   "Unit1.MotionNodes".PLCToMotion.Parameters.StackMain.StackCalculate.TeachingPos.StartPos.CathodePnPX1 := "Unit1.Em5.Config".cmCathodeMainPnP1AxisX.setPositions[0].position;
   "Unit1.MotionNodes".PLCToMotion.Parameters.StackMain.StackCalculate.TeachingPos.StartPos.CathodePnPX2 := "Unit1.Em5.Config".cmCathodeMainPnP2AxisX.setPositions[0].position;
   "Unit1.MotionNodes".PLCToMotion.Parameters.StackMain.StackCalculate.TeachingPos.StartPos.CathodePnPZ1 := "Unit1.Em5.Config".cmCathodeMainPnP1AxisZ.setPositions[0].position;
   "Unit1.MotionNodes".PLCToMotion.Parameters.StackMain.StackCalculate.TeachingPos.StartPos.CathodePnPZ2 := "Unit1.Em5.Config".cmCathodeMainPnP2AxisZ.setPositions[0].position;

   "Unit1.MotionNodes".PLCToMotion.Parameters.StackMain.StackCalculate.TeachingPos.StartPos.AnodeMandrelYFront := "Unit1.Em6.Config".cmMendrelAnodeFrontAxisY.setPositions[0].position;
   "Unit1.MotionNodes".PLCToMotion.Parameters.StackMain.StackCalculate.TeachingPos.StartPos.AnodeMandrelYRear := "Unit1.Em6.Config".cmMendrelAnodeRearAxisY.setPositions[0].position;
   "Unit1.MotionNodes".PLCToMotion.Parameters.StackMain.StackCalculate.TeachingPos.StartPos.AnodeMandrelZFront := "Unit1.Em6.Config".cmMendrelAnodeFrontAxisZ.setPositions[0].position;
   "Unit1.MotionNodes".PLCToMotion.Parameters.StackMain.StackCalculate.TeachingPos.StartPos.AnodeMandrelZRear := "Unit1.Em6.Config".cmMendrelAnodeRearAxisZ.setPositions[0].position;
   "Unit1.MotionNodes".PLCToMotion.Parameters.StackMain.StackCalculate.TeachingPos.StartPos.CathodeMandrelYFront := "Unit1.Em6.Config".cmMendrelCathodeFrontAxisY.setPositions[0].position;
   "Unit1.MotionNodes".PLCToMotion.Parameters.StackMain.StackCalculate.TeachingPos.StartPos.CathodeMandrelYRear := "Unit1.Em6.Config".cmMendrelCathodeRearAxisY.setPositions[0].position;
   "Unit1.MotionNodes".PLCToMotion.Parameters.StackMain.StackCalculate.TeachingPos.StartPos.CathodeMandrelZFront := "Unit1.Em6.Config".cmMendrelCathodeFrontAxisZ.setPositions[0].position;
   "Unit1.MotionNodes".PLCToMotion.Parameters.StackMain.StackCalculate.TeachingPos.StartPos.CathodeMandrelZRear := "Unit1.Em6.Config".cmMendrelCathodeRearAxisZ.setPositions[0].position;

   ///// End Pos

   "Unit1.MotionNodes".PLCToMotion.Parameters.StackMain.StackCalculate.TeachingPos.EndPos.FinalRoller := "Unit1.Em6.Config".cmFinalRollerFrontAxisX.setPositions[1].position;
   "Unit1.MotionNodes".PLCToMotion.Parameters.StackMain.StackCalculate.TeachingPos.EndPos.AnodePnPX1 := "Unit1.Em4.Config".cmAnodeMainPnP1AxisX.setPositions[1].position;
   "Unit1.MotionNodes".PLCToMotion.Parameters.StackMain.StackCalculate.TeachingPos.EndPos.AnodePnPX2 := "Unit1.Em4.Config".cmAnodeMainPnP2AxisX.setPositions[1].position;

   "Unit1.MotionNodes".PLCToMotion.Parameters.StackMain.StackCalculate.TeachingPos.EndPos.AnodePnPZ1P1 := "Unit1.Em4.Config".cmAnodeMainPnP1AxisZ.setPositions[1].position;
   "Unit1.MotionNodes".PLCToMotion.Parameters.StackMain.StackCalculate.TeachingPos.EndPos.AnodePnPZ1P2 := "Unit1.Em4.Config".cmAnodeMainPnP1AxisZ.setPositions[2].position;
   "Unit1.MotionNodes".PLCToMotion.Parameters.StackMain.StackCalculate.TeachingPos.EndPos.AnodePnPZ2P1 := "Unit1.Em4.Config".cmAnodeMainPnP2AxisZ.setPositions[1].position;
   "Unit1.MotionNodes".PLCToMotion.Parameters.StackMain.StackCalculate.TeachingPos.EndPos.AnodePnPZ2P2 := "Unit1.Em4.Config".cmAnodeMainPnP2AxisZ.setPositions[2].position;

   "Unit1.MotionNodes".PLCToMotion.Parameters.StackMain.StackCalculate.TeachingPos.EndPos.CathodePnPX1 := "Unit1.Em5.Config".cmCathodeMainPnP1AxisX.setPositions[1].position;
   "Unit1.MotionNodes".PLCToMotion.Parameters.StackMain.StackCalculate.TeachingPos.EndPos.CathodePnPX2 := "Unit1.Em5.Config".cmCathodeMainPnP2AxisX.setPositions[1].position;

   "Unit1.MotionNodes".PLCToMotion.Parameters.StackMain.StackCalculate.TeachingPos.EndPos.CathodePnPZ1P1 := "Unit1.Em5.Config".cmCathodeMainPnP1AxisZ.setPositions[1].position;
   "Unit1.MotionNodes".PLCToMotion.Parameters.StackMain.StackCalculate.TeachingPos.EndPos.CathodePnPZ1P2 := "Unit1.Em5.Config".cmCathodeMainPnP1AxisZ.setPositions[2].position;
   "Unit1.MotionNodes".PLCToMotion.Parameters.StackMain.StackCalculate.TeachingPos.EndPos.CathodePnPZ2P1 := "Unit1.Em5.Config".cmCathodeMainPnP2AxisZ.setPositions[1].position;
   "Unit1.MotionNodes".PLCToMotion.Parameters.StackMain.StackCalculate.TeachingPos.EndPos.CathodePnPZ2P2 := "Unit1.Em5.Config".cmCathodeMainPnP2AxisZ.setPositions[2].position;


   "Unit1.MotionNodes".PLCToMotion.Parameters.StackMain.StackCalculate.TeachingPos.EndPos.AnodeMandrelYFront := "Unit1.Em6.Config".cmMendrelAnodeFrontAxisY.setPositions[1].position;
   "Unit1.MotionNodes".PLCToMotion.Parameters.StackMain.StackCalculate.TeachingPos.EndPos.AnodeMandrelYRear := "Unit1.Em6.Config".cmMendrelAnodeRearAxisY.setPositions[1].position;
   "Unit1.MotionNodes".PLCToMotion.Parameters.StackMain.StackCalculate.TeachingPos.EndPos.AnodeMandrelZFront := "Unit1.Em6.Config".cmMendrelAnodeFrontAxisZ.setPositions[1].position;
   "Unit1.MotionNodes".PLCToMotion.Parameters.StackMain.StackCalculate.TeachingPos.EndPos.AnodeMandrelZRear := "Unit1.Em6.Config".cmMendrelAnodeRearAxisZ.setPositions[1].position;
   "Unit1.MotionNodes".PLCToMotion.Parameters.StackMain.StackCalculate.TeachingPos.EndPos.CathodeMandrelYFront := "Unit1.Em6.Config".cmMendrelCathodeFrontAxisY.setPositions[1].position;
   "Unit1.MotionNodes".PLCToMotion.Parameters.StackMain.StackCalculate.TeachingPos.EndPos.CathodeMandrelYRear := "Unit1.Em6.Config".cmMendrelCathodeRearAxisY.setPositions[1].position;
   "Unit1.MotionNodes".PLCToMotion.Parameters.StackMain.StackCalculate.TeachingPos.EndPos.CathodeMandrelZFront := "Unit1.Em6.Config".cmMendrelCathodeFrontAxisZ.setPositions[1].position;
   "Unit1.MotionNodes".PLCToMotion.Parameters.StackMain.StackCalculate.TeachingPos.EndPos.CathodeMandrelZRear := "Unit1.Em6.Config".cmMendrelCathodeRearAxisZ.setPositions[1].position;
END_REGION

REGION Network 8 (SCL): PLC -> HMI Softcam
   "HMI_Interface_Parameter".Softcam[1] := "Unit1.Em0.HmiInterface".cm.softCam.unwinderTopAxisB;
   "HMI_Interface_Parameter".Softcam[2] := "Unit1.Em1.HmiInterface".cm.softCam.unwinderBtmAxisB;
   "HMI_Interface_Parameter".Softcam[3] := "Unit1.Em3.HmiInterface".cm.softCam.compensatorAxisX;
   "HMI_Interface_Parameter".Softcam[4] := "Unit1.Em7.HmiInterface".cm.softCam.jrPusherAxisZ;
   "HMI_Interface_Parameter".Softcam[5] := "Unit1.Em4.HmiInterface".cm.softCam.anodeMainPnP1AxisX;
   "HMI_Interface_Parameter".Softcam[6] := "Unit1.Em4.HmiInterface".cm.softCam.anodeMainPnP2AxisX;
   "HMI_Interface_Parameter".Softcam[7] := "Unit1.Em5.HmiInterface".cm.softCam.cathodeMainPnP1AxisX;
   "HMI_Interface_Parameter".Softcam[8] := "Unit1.Em5.HmiInterface".cm.softCam.cathodeMainPnP2AxisX;
   "HMI_Interface_Parameter".Softcam[9] := "Unit1.Em5.HmiInterface".cm.softCam.cathodeMainPnP1AxisY;
   "HMI_Interface_Parameter".Softcam[10] := "Unit1.Em5.HmiInterface".cm.softCam.cathodeMainPnP1AxisZ;
   "HMI_Interface_Parameter".Softcam[11] := "Unit1.Em4.HmiInterface".cm.softCam.anodeMainPnP1AxisY;
   "HMI_Interface_Parameter".Softcam[12] := "Unit1.Em4.HmiInterface".cm.softCam.anodeMainPnP1AxisZ;
   "HMI_Interface_Parameter".Softcam[13] := "Unit1.Em5.HmiInterface".cm.softCam.cathodeMainPnP2AxisZ;
   "HMI_Interface_Parameter".Softcam[14] := "Unit1.Em4.HmiInterface".cm.softCam.anodeMainPnP2AxisZ;
   "HMI_Interface_Parameter".Softcam[15] := "Unit1.Em4.HmiInterface".cm.softCam.anodeAlignTableAxisX;
   "HMI_Interface_Parameter".Softcam[16] := "Unit1.Em4.HmiInterface".cm.softCam.anodeAlignTableAxisY2;
   "HMI_Interface_Parameter".Softcam[17] := "Unit1.Em4.HmiInterface".cm.softCam.anodeAlignTableAxisY1;
   "HMI_Interface_Parameter".Softcam[18] := "Unit1.Em5.HmiInterface".cm.softCam.cathodeAlignTableAxisX;
   "HMI_Interface_Parameter".Softcam[19] := "Unit1.Em5.HmiInterface".cm.softCam.cathodeAlignTableAxisY2;
   "HMI_Interface_Parameter".Softcam[20] := "Unit1.Em5.HmiInterface".cm.softCam.cathodeAlignTableAxisY1;
   "HMI_Interface_Parameter".Softcam[21] := "Unit1.Em6.HmiInterface".cm.softCam.finalRollerFrontAxisX;
   "HMI_Interface_Parameter".Softcam[22] := "Unit1.Em6.HmiInterface".cm.softCam.finalRollerRearAxisX;
   "HMI_Interface_Parameter".Softcam[23] := "Unit1.Em6.HmiInterface".cm.softCam.mendrelAnodeFrontAxisY;
   "HMI_Interface_Parameter".Softcam[24] := "Unit1.Em6.HmiInterface".cm.softCam.mendrelAnodeFrontAxisZ;
   "HMI_Interface_Parameter".Softcam[25] := "Unit1.Em6.HmiInterface".cm.softCam.mendrelAnodeRearAxisY;
   "HMI_Interface_Parameter".Softcam[26] := "Unit1.Em6.HmiInterface".cm.softCam.mendrelAnodeRearAxisZ;
   "HMI_Interface_Parameter".Softcam[27] := "Unit1.Em6.HmiInterface".cm.softCam.mendrelCathodeFrontAxisY;
   "HMI_Interface_Parameter".Softcam[28] := "Unit1.Em6.HmiInterface".cm.softCam.mendrelCathodeFrontAxisZ;
   "HMI_Interface_Parameter".Softcam[29] := "Unit1.Em6.HmiInterface".cm.softCam.mendrelCathodeRearAxisY;
   "HMI_Interface_Parameter".Softcam[30] := "Unit1.Em6.HmiInterface".cm.softCam.mendrelCathodeRearAxisZ;
   "HMI_Interface_Parameter".Softcam[31] := "Unit1.Em6.HmiInterface".cm.softCam.stackTableAxisZ;
   "HMI_Interface_Parameter".Softcam[32] := "Unit1.Em6.HmiInterface".cm.softCam.stackTableOutFrontAxisZ;
   "HMI_Interface_Parameter".Softcam[33] := "Unit1.Em6.HmiInterface".cm.softCam.stackTableOutRearAxisZ;
   "HMI_Interface_Parameter".Softcam[34] := "Unit1.Em7.HmiInterface".cm.softCam.sepaClampnCutterAxisX;
   "HMI_Interface_Parameter".Softcam[35] := "Unit1.Em7.HmiInterface".cm.softCam.sepaClampnCutterAxisZ;
   "HMI_Interface_Parameter".Softcam[36] := "Unit1.Em7.HmiInterface".cm.softCam.sepaGripperAxisX;
   "HMI_Interface_Parameter".Softcam[37] := "Unit1.Em7.HmiInterface".cm.softCam.sepaGripperAxisZ;
   "HMI_Interface_Parameter".Softcam[38] := "Unit1.Em7.HmiInterface".cm.softCam.sepaGripperAxisC;
   "HMI_Interface_Parameter".Softcam[39] := "Unit1.Em7.HmiInterface".cm.softCam.jrWinderRearAxisY;
   "HMI_Interface_Parameter".Softcam[40] := "Unit1.Em7.HmiInterface".cm.softCam.jrWinderFrontAxisY;
   "HMI_Interface_Parameter".Softcam[41] := "Unit1.Em7.HmiInterface".cm.softCam.jrWinderAxisB;
END_REGION

REGION Network 9 (SCL): SamplingMode Complete end
   IF "Unit1.EmNodes".SamplingModeComplete THEN
       "HMI_Interface_Parameter".FATModeInterface.ModeSelect.SamplingMode := FALSE;
       ;
   END_IF;
END_REGION

REGION Network 10: SamplingMode Btn on count reset trigger // cell current count
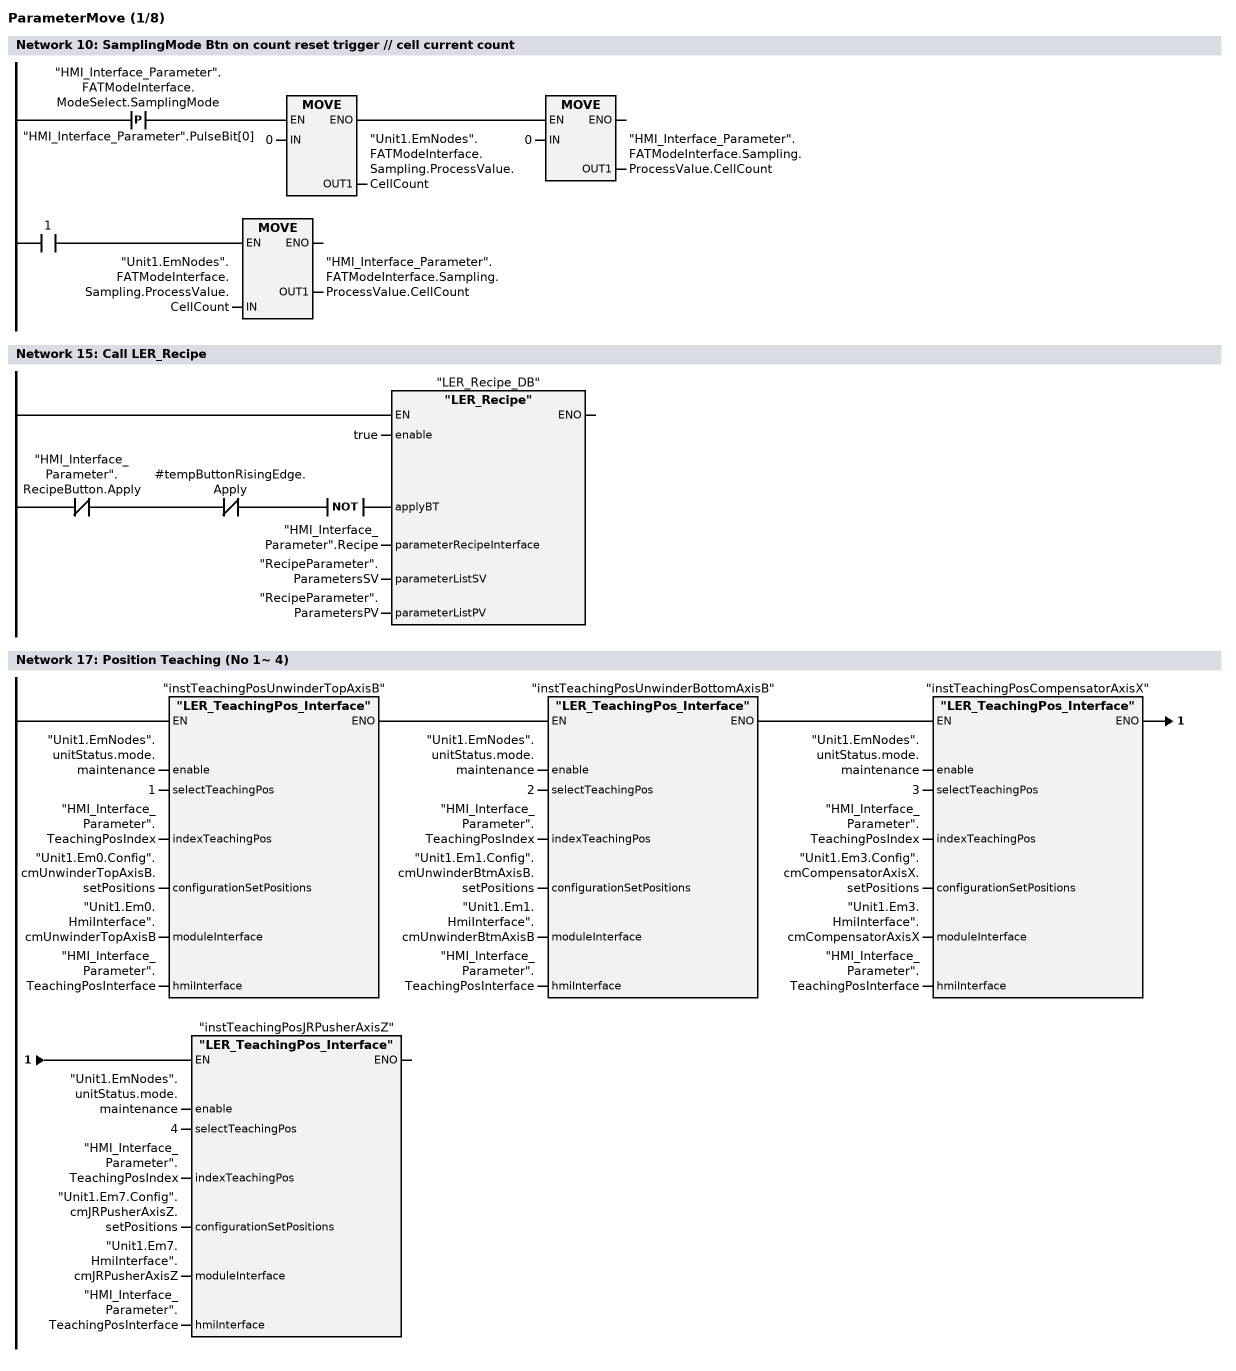
   RUNG wire#powerrail
      P_Contact(operand := "HMI_Interface_Parameter".FATModeInterface.ModeSelect.SamplingMode, bit := "HMI_Interface_Parameter".PulseBit[0])
      Move(in := 0, out1 => "Unit1.EmNodes".FATModeInterface.Sampling.ProcessValue.CellCount)
      Move(in := 0, out1 => "HMI_Interface_Parameter".FATModeInterface.Sampling.ProcessValue.CellCount)
   END_RUNG
   RUNG wire#powerrail
      Contact( 1 )
      Move(in := "Unit1.EmNodes".FATModeInterface.Sampling.ProcessValue.CellCount, out1 => "HMI_Interface_Parameter".FATModeInterface.Sampling.ProcessValue.CellCount)
   END_RUNG
   // the same network as SCL:
   #_w1 := "HMI_Interface_Parameter".FATModeInterface.ModeSelect.SamplingMode AND NOT "HMI_Interface_Parameter".PulseBit[0];   // rising edge of "HMI_Interface_Parameter".FATModeInterface.ModeSelect.SamplingMode
   "HMI_Interface_Parameter".PulseBit[0] := "HMI_Interface_Parameter".FATModeInterface.ModeSelect.SamplingMode;
   IF #_w1 THEN
       "Unit1.EmNodes".FATModeInterface.Sampling.ProcessValue.CellCount := 0;
       "HMI_Interface_Parameter".FATModeInterface.Sampling.ProcessValue.CellCount := 0;
   END_IF;
   IF 1 THEN
       "HMI_Interface_Parameter".FATModeInterface.Sampling.ProcessValue.CellCount := "Unit1.EmNodes".FATModeInterface.Sampling.ProcessValue.CellCount;
   END_IF;
END_REGION

REGION Network 12 (SCL): HMI Interface Parameter To Recipe Pareameter SV
   // IF #tempButtonRisingEdge.Apply THEN
   //     "RecipeParameter".ParametersSV.Recipe1 := "HMI_Interface_Parameter"."Default Recipe".SetValue."Electrode Width".Anode;
   //     "RecipeParameter".ParametersSV.Recipe2 := "HMI_Interface_Parameter"."Default Recipe".SetValue."Electrode Width".Cathode;
   //     "RecipeParameter".ParametersSV.Recipe3 := "HMI_Interface_Parameter"."Default Recipe".SetValue."Anode Thinkness";
   //     "RecipeParameter".ParametersSV.Recipe4 := "HMI_Interface_Parameter"."Default Recipe".SetValue."Cathode Thinkness";
   //     "RecipeParameter".ParametersSV.Recipe5 := "HMI_Interface_Parameter"."Default Recipe".SetValue."Sperator Thinkness";
   //     "RecipeParameter".ParametersSV.Recipe6 := "HMI_Interface_Parameter"."Default Recipe".SetValue."Jelly Roll Width";
   //     "RecipeParameter".ParametersSV.Recipe7 := "HMI_Interface_Parameter"."Default Recipe".SetValue."Cell Stack Count";
   //     "RecipeParameter".ParametersSV.Recipe8 := "HMI_Interface_Parameter".Parameter_Image[0]."Set Value";
   //     "RecipeParameter".ParametersSV.Recipe9 := "HMI_Interface_Parameter".Parameter_Image[1]."Set Value";
   //     //
   //     //"RecipeParameter".ParametersSV.Recipe10 := ;
   //     //"RecipeParameter".ParametersSV.Recipe11 := ;
   //     //"RecipeParameter".ParametersSV.Recipe12 := ;
   //     //"RecipeParameter".ParametersSV.Recipe13 := ;
   //     //"RecipeParameter".ParametersSV.Recipe14 := ;
   //     //"RecipeParameter".ParametersSV.Recipe15 := ;
   //     //"RecipeParameter".ParametersSV.Recipe16 := ;
   //     //"RecipeParameter".ParametersSV.Recipe17 := ;
   //     //"RecipeParameter".ParametersSV.Recipe18 := ;
   //     //"RecipeParameter".ParametersSV.Recipe19 := ;
   //     //"RecipeParameter".ParametersSV.Recipe20 := ;
   //     //"RecipeParameter".ParametersSV.Recipe21 := ;
   //     //"RecipeParameter".ParametersSV.Recipe22 := ;
   //     //"RecipeParameter".ParametersSV.Recipe23 := ;
   //     //"RecipeParameter".ParametersSV.Recipe24 := ;
   //     //"RecipeParameter".ParametersSV.Recipe25 := ;
   // END_IF;
END_REGION

REGION Network 13 (SCL): HMI Interface Pareameter Recipe Data To HMI Interface Parameter Process Value
   // IF "HMI_Interface_Parameter".Recipe.RecipeChangeBT OR "HMI_Interface_Parameter".RecipeButton.Apply OR #tempButtonRisingEdge.Apply THEN

   //     "HMI_Interface_Parameter"."Default Recipe".ProcessValue."Electrode Width".Anode := "HMI_Interface_Parameter".Recipe.Recipe_Data["HMI_Interface_Parameter".Recipe.CurrentRecipeNum].Recipe1;
   //     "HMI_Interface_Parameter"."Default Recipe".ProcessValue."Electrode Width".Cathode := "HMI_Interface_Parameter".Recipe.Recipe_Data["HMI_Interface_Parameter".Recipe.CurrentRecipeNum].Recipe2;
   //     "HMI_Interface_Parameter"."Default Recipe".ProcessValue."Anode Thinkness" := "HMI_Interface_Parameter".Recipe.Recipe_Data["HMI_Interface_Parameter".Recipe.CurrentRecipeNum].Recipe3;
   //     "HMI_Interface_Parameter"."Default Recipe".ProcessValue."Cathode Thinkness" := "HMI_Interface_Parameter".Recipe.Recipe_Data["HMI_Interface_Parameter".Recipe.CurrentRecipeNum].Recipe4;
   //     "HMI_Interface_Parameter"."Default Recipe".ProcessValue."Sperator Thinkness" := "HMI_Interface_Parameter".Recipe.Recipe_Data["HMI_Interface_Parameter".Recipe.CurrentRecipeNum].Recipe5;
   //     "HMI_Interface_Parameter"."Default Recipe".ProcessValue."Jelly Roll Width" := "HMI_Interface_Parameter".Recipe.Recipe_Data["HMI_Interface_Parameter".Recipe.CurrentRecipeNum].Recipe6;
   //     "HMI_Interface_Parameter"."Default Recipe".ProcessValue."Cell Stack Count" := LREAL_TO_SINT("HMI_Interface_Parameter".Recipe.Recipe_Data["HMI_Interface_Parameter".Recipe.CurrentRecipeNum].Recipe7);
   //     "HMI_Interface_Parameter".Parameter_Image[0]."Process Value" := "HMI_Interface_Parameter".Recipe.Recipe_Data["HMI_Interface_Parameter".Recipe.CurrentRecipeNum].Recipe8;
   //     "HMI_Interface_Parameter".Parameter_Image[1]."Process Value" := "HMI_Interface_Parameter".Recipe.Recipe_Data["HMI_Interface_Parameter".Recipe.CurrentRecipeNum].Recipe9;
   //     // := "HMI_Interface_Parameter".Recipe.Recipe_Data["HMI_Interface_Parameter".Recipe.CurrentRecipeNum].Recipe10;
   //     // := "HMI_Interface_Parameter".Recipe.Recipe_Data["HMI_Interface_Parameter".Recipe.CurrentRecipeNum].Recipe11;
   //     // := "HMI_Interface_Parameter".Recipe.Recipe_Data["HMI_Interface_Parameter".Recipe.CurrentRecipeNum].Recipe12;
   //     // := "HMI_Interface_Parameter".Recipe.Recipe_Data["HMI_Interface_Parameter".Recipe.CurrentRecipeNum].Recipe13;
   //     // := "HMI_Interface_Parameter".Recipe.Recipe_Data["HMI_Interface_Parameter".Recipe.CurrentRecipeNum].Recipe14;
   //     // := "HMI_Interface_Parameter".Recipe.Recipe_Data["HMI_Interface_Parameter".Recipe.CurrentRecipeNum].Recipe15;
   // END_IF;
END_REGION

REGION Network 14 (SCL): Recipe Parameter PV To Unit EmData Recipe
   "Unit1.EmData".UnitRecipe.size.Anode.length := "RecipeParameter".ParametersPV.Recipe1;
   "Unit1.EmData".UnitRecipe.size.Cathode.length := "RecipeParameter".ParametersPV.Recipe2;
   "Unit1.EmData".UnitRecipe.size.Anode.thickness := "RecipeParameter".ParametersPV.Recipe3;
   "Unit1.EmData".UnitRecipe.size.Cathode.thickness := "RecipeParameter".ParametersPV.Recipe4;
   "Unit1.EmData".UnitRecipe.SepaThickness := "RecipeParameter".ParametersPV.Recipe5;
   "Unit1.EmData".UnitRecipe.JellyRollWidth := "RecipeParameter".ParametersPV.Recipe6;
   "Unit1.EmData".UnitRecipe.StackCount := "RecipeParameter".ParametersPV.Recipe7;
   "Unit1.EmData".UnitRecipe.DancerRegulator := "RecipeParameter".ParametersPV.Recipe8;
   "Unit1.EmData".UnitRecipe.AutoSpliceRemainingLength := "RecipeParameter".ParametersPV.Recipe9;
   //
   // := "RecipeParameter".ParametersPV.Recipe10;
   // := "RecipeParameter".ParametersPV.Recipe11;
   // := "RecipeParameter".ParametersPV.Recipe12;
   // := "RecipeParameter".ParametersPV.Recipe13;
   // := "RecipeParameter".ParametersPV.Recipe14;
   // := "RecipeParameter".ParametersPV.Recipe15;
END_REGION

REGION Network 15: Call LER_Recipe
   RUNG wire#powerrail
      "LER_Recipe_DB"(applyBT := wire#w1, enable := true, parameterRecipeInterface := "HMI_Interface_Parameter".Recipe, parameterListSV := "RecipeParameter".ParametersSV, parameterListPV := "RecipeParameter".ParametersPV)
   END_RUNG
   RUNG wire#powerrail
      I_Contact( "HMI_Interface_Parameter".RecipeButton.Apply )
      I_Contact( #tempButtonRisingEdge.Apply )
      Not()
   END_RUNG wire#w1
   // the same network as SCL:
   "LER_Recipe_DB"(enable := true,   // "LER_Recipe"
                   applyBT := NOT (NOT "HMI_Interface_Parameter".RecipeButton.Apply AND NOT #tempButtonRisingEdge.Apply),
                   parameterRecipeInterface := "HMI_Interface_Parameter".Recipe,
                   parameterListSV := "RecipeParameter".ParametersSV,
                   parameterListPV := "RecipeParameter".ParametersPV);
END_REGION

REGION Network 17: Position Teaching (No 1~ 4)
   RUNG wire#powerrail
      "instTeachingPosUnwinderTopAxisB"(enable := "Unit1.EmNodes".unitStatus.mode.maintenance, selectTeachingPos := 1, indexTeachingPos := "HMI_Interface_Parameter".TeachingPosIndex, configurationSetPositions := "Unit1.Em0.Config".cmUnwinderTopAxisB.setPositions, moduleInterface := "Unit1.Em0.HmiInterface".cmUnwinderTopAxisB, hmiInterface := "HMI_Interface_Parameter".TeachingPosInterface)
      "instTeachingPosUnwinderBottomAxisB"(enable := "Unit1.EmNodes".unitStatus.mode.maintenance, selectTeachingPos := 2, indexTeachingPos := "HMI_Interface_Parameter".TeachingPosIndex, configurationSetPositions := "Unit1.Em1.Config".cmUnwinderBtmAxisB.setPositions, moduleInterface := "Unit1.Em1.HmiInterface".cmUnwinderBtmAxisB, hmiInterface := "HMI_Interface_Parameter".TeachingPosInterface)
      "instTeachingPosCompensatorAxisX"(enable := "Unit1.EmNodes".unitStatus.mode.maintenance, selectTeachingPos := 3, indexTeachingPos := "HMI_Interface_Parameter".TeachingPosIndex, configurationSetPositions := "Unit1.Em3.Config".cmCompensatorAxisX.setPositions, moduleInterface := "Unit1.Em3.HmiInterface".cmCompensatorAxisX, hmiInterface := "HMI_Interface_Parameter".TeachingPosInterface)
      "instTeachingPosJRPusherAxisZ"(enable := "Unit1.EmNodes".unitStatus.mode.maintenance, selectTeachingPos := 4, indexTeachingPos := "HMI_Interface_Parameter".TeachingPosIndex, configurationSetPositions := "Unit1.Em7.Config".cmJRPusherAxisZ.setPositions, moduleInterface := "Unit1.Em7.HmiInterface".cmJRPusherAxisZ, hmiInterface := "HMI_Interface_Parameter".TeachingPosInterface)
   END_RUNG
   // the same network as SCL:
   "instTeachingPosUnwinderTopAxisB"(enable := "Unit1.EmNodes".unitStatus.mode.maintenance,   // "LER_TeachingPos_Interface"
                           selectTeachingPos := 1,
                           indexTeachingPos := "HMI_Interface_Parameter".TeachingPosIndex,
                           configurationSetPositions := "Unit1.Em0.Config".cmUnwinderTopAxisB.setPositions,
                           moduleInterface := "Unit1.Em0.HmiInterface".cmUnwinderTopAxisB,
                           hmiInterface := "HMI_Interface_Parameter".TeachingPosInterface,
                           ENO => #_w1);
   "instTeachingPosUnwinderBottomAxisB"(EN := #_w1,   // "LER_TeachingPos_Interface"
                           enable := "Unit1.EmNodes".unitStatus.mode.maintenance,
                           selectTeachingPos := 2,
                           indexTeachingPos := "HMI_Interface_Parameter".TeachingPosIndex,
                           configurationSetPositions := "Unit1.Em1.Config".cmUnwinderBtmAxisB.setPositions,
                           moduleInterface := "Unit1.Em1.HmiInterface".cmUnwinderBtmAxisB,
                           hmiInterface := "HMI_Interface_Parameter".TeachingPosInterface,
                           ENO => #_w2);
   "instTeachingPosCompensatorAxisX"(EN := #_w2,   // "LER_TeachingPos_Interface"
                           enable := "Unit1.EmNodes".unitStatus.mode.maintenance,
                           selectTeachingPos := 3,
                           indexTeachingPos := "HMI_Interface_Parameter".TeachingPosIndex,
                           configurationSetPositions := "Unit1.Em3.Config".cmCompensatorAxisX.setPositions,
                           moduleInterface := "Unit1.Em3.HmiInterface".cmCompensatorAxisX,
                           hmiInterface := "HMI_Interface_Parameter".TeachingPosInterface,
                           ENO => #_w3);
   IF #_w3 THEN
       "instTeachingPosJRPusherAxisZ"(enable := "Unit1.EmNodes".unitStatus.mode.maintenance,   // "LER_TeachingPos_Interface"
                               selectTeachingPos := 4,
                               indexTeachingPos := "HMI_Interface_Parameter".TeachingPosIndex,
                               configurationSetPositions := "Unit1.Em7.Config".cmJRPusherAxisZ.setPositions,
                               moduleInterface := "Unit1.Em7.HmiInterface".cmJRPusherAxisZ,
                               hmiInterface := "HMI_Interface_Parameter".TeachingPosInterface);
   END_IF;
END_REGION

REGION Network 18: Position Teaching (No 5~8)
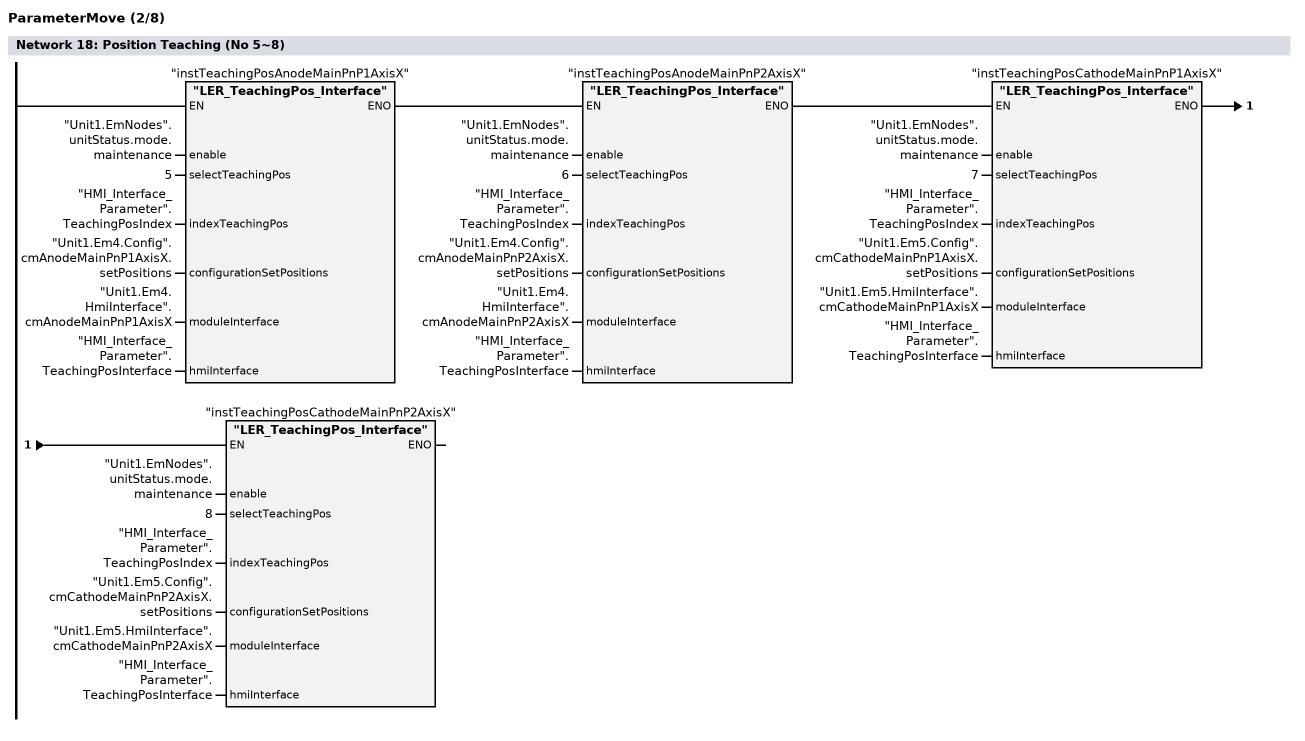
   RUNG wire#powerrail
      "instTeachingPosAnodeMainPnP1AxisX"(enable := "Unit1.EmNodes".unitStatus.mode.maintenance, selectTeachingPos := 5, indexTeachingPos := "HMI_Interface_Parameter".TeachingPosIndex, configurationSetPositions := "Unit1.Em4.Config".cmAnodeMainPnP1AxisX.setPositions, moduleInterface := "Unit1.Em4.HmiInterface".cmAnodeMainPnP1AxisX, hmiInterface := "HMI_Interface_Parameter".TeachingPosInterface)
      "instTeachingPosAnodeMainPnP2AxisX"(enable := "Unit1.EmNodes".unitStatus.mode.maintenance, selectTeachingPos := 6, indexTeachingPos := "HMI_Interface_Parameter".TeachingPosIndex, configurationSetPositions := "Unit1.Em4.Config".cmAnodeMainPnP2AxisX.setPositions, moduleInterface := "Unit1.Em4.HmiInterface".cmAnodeMainPnP2AxisX, hmiInterface := "HMI_Interface_Parameter".TeachingPosInterface)
      "instTeachingPosCathodeMainPnP1AxisX"(enable := "Unit1.EmNodes".unitStatus.mode.maintenance, selectTeachingPos := 7, indexTeachingPos := "HMI_Interface_Parameter".TeachingPosIndex, configurationSetPositions := "Unit1.Em5.Config".cmCathodeMainPnP1AxisX.setPositions, moduleInterface := "Unit1.Em5.HmiInterface".cmCathodeMainPnP1AxisX, hmiInterface := "HMI_Interface_Parameter".TeachingPosInterface)
      "instTeachingPosCathodeMainPnP2AxisX"(enable := "Unit1.EmNodes".unitStatus.mode.maintenance, selectTeachingPos := 8, indexTeachingPos := "HMI_Interface_Parameter".TeachingPosIndex, configurationSetPositions := "Unit1.Em5.Config".cmCathodeMainPnP2AxisX.setPositions, moduleInterface := "Unit1.Em5.HmiInterface".cmCathodeMainPnP2AxisX, hmiInterface := "HMI_Interface_Parameter".TeachingPosInterface)
   END_RUNG
   // the same network as SCL:
   "instTeachingPosAnodeMainPnP1AxisX"(enable := "Unit1.EmNodes".unitStatus.mode.maintenance,   // "LER_TeachingPos_Interface"
                           selectTeachingPos := 5,
                           indexTeachingPos := "HMI_Interface_Parameter".TeachingPosIndex,
                           configurationSetPositions := "Unit1.Em4.Config".cmAnodeMainPnP1AxisX.setPositions,
                           moduleInterface := "Unit1.Em4.HmiInterface".cmAnodeMainPnP1AxisX,
                           hmiInterface := "HMI_Interface_Parameter".TeachingPosInterface,
                           ENO => #_w1);
   "instTeachingPosAnodeMainPnP2AxisX"(EN := #_w1,   // "LER_TeachingPos_Interface"
                           enable := "Unit1.EmNodes".unitStatus.mode.maintenance,
                           selectTeachingPos := 6,
                           indexTeachingPos := "HMI_Interface_Parameter".TeachingPosIndex,
                           configurationSetPositions := "Unit1.Em4.Config".cmAnodeMainPnP2AxisX.setPositions,
                           moduleInterface := "Unit1.Em4.HmiInterface".cmAnodeMainPnP2AxisX,
                           hmiInterface := "HMI_Interface_Parameter".TeachingPosInterface,
                           ENO => #_w2);
   "instTeachingPosCathodeMainPnP1AxisX"(EN := #_w2,   // "LER_TeachingPos_Interface"
                           enable := "Unit1.EmNodes".unitStatus.mode.maintenance,
                           selectTeachingPos := 7,
                           indexTeachingPos := "HMI_Interface_Parameter".TeachingPosIndex,
                           configurationSetPositions := "Unit1.Em5.Config".cmCathodeMainPnP1AxisX.setPositions,
                           moduleInterface := "Unit1.Em5.HmiInterface".cmCathodeMainPnP1AxisX,
                           hmiInterface := "HMI_Interface_Parameter".TeachingPosInterface,
                           ENO => #_w3);
   IF #_w3 THEN
       "instTeachingPosCathodeMainPnP2AxisX"(enable := "Unit1.EmNodes".unitStatus.mode.maintenance,   // "LER_TeachingPos_Interface"
                               selectTeachingPos := 8,
                               indexTeachingPos := "HMI_Interface_Parameter".TeachingPosIndex,
                               configurationSetPositions := "Unit1.Em5.Config".cmCathodeMainPnP2AxisX.setPositions,
                               moduleInterface := "Unit1.Em5.HmiInterface".cmCathodeMainPnP2AxisX,
                               hmiInterface := "HMI_Interface_Parameter".TeachingPosInterface);
   END_IF;
END_REGION

REGION Network 19: Position Teaching (No 9~12)
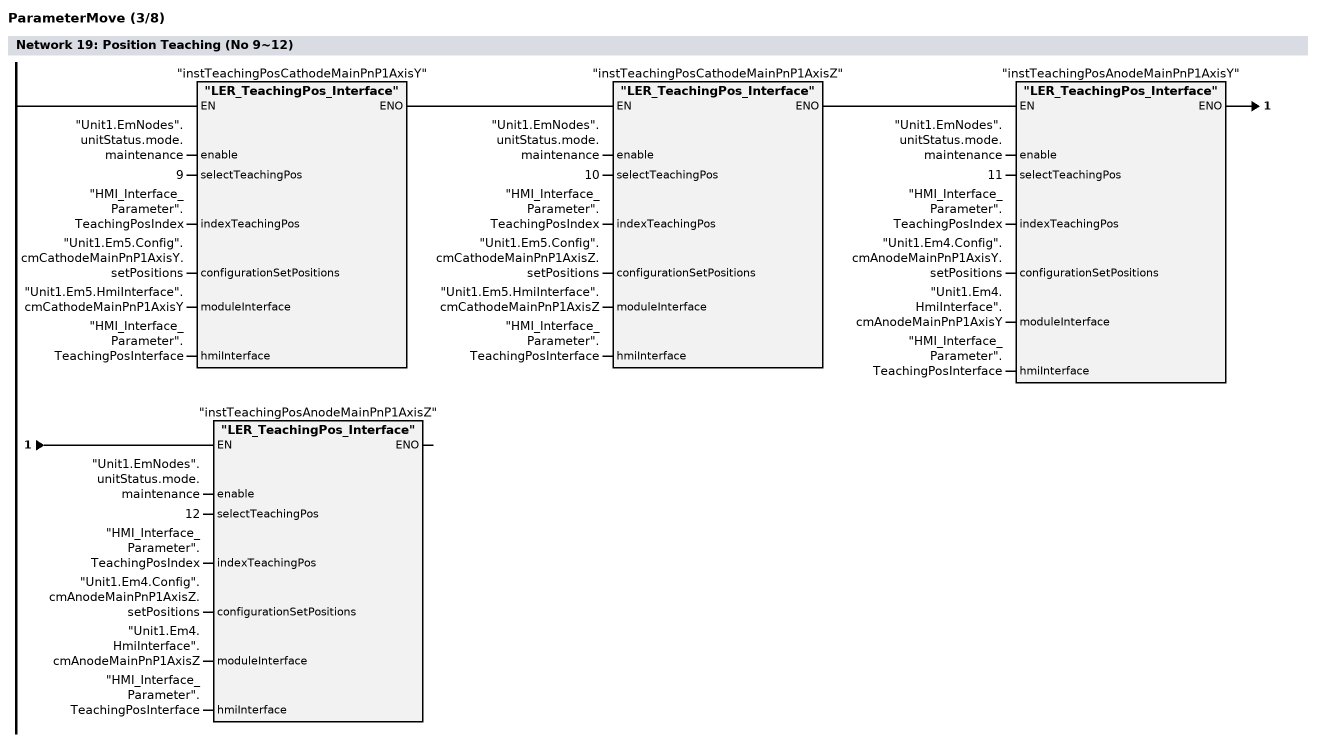
   RUNG wire#powerrail
      "instTeachingPosCathodeMainPnP1AxisY"(enable := "Unit1.EmNodes".unitStatus.mode.maintenance, selectTeachingPos := 9, indexTeachingPos := "HMI_Interface_Parameter".TeachingPosIndex, configurationSetPositions := "Unit1.Em5.Config".cmCathodeMainPnP1AxisY.setPositions, moduleInterface := "Unit1.Em5.HmiInterface".cmCathodeMainPnP1AxisY, hmiInterface := "HMI_Interface_Parameter".TeachingPosInterface)
      "instTeachingPosCathodeMainPnP1AxisZ"(enable := "Unit1.EmNodes".unitStatus.mode.maintenance, selectTeachingPos := 10, indexTeachingPos := "HMI_Interface_Parameter".TeachingPosIndex, configurationSetPositions := "Unit1.Em5.Config".cmCathodeMainPnP1AxisZ.setPositions, moduleInterface := "Unit1.Em5.HmiInterface".cmCathodeMainPnP1AxisZ, hmiInterface := "HMI_Interface_Parameter".TeachingPosInterface)
      "instTeachingPosAnodeMainPnP1AxisY"(enable := "Unit1.EmNodes".unitStatus.mode.maintenance, selectTeachingPos := 11, indexTeachingPos := "HMI_Interface_Parameter".TeachingPosIndex, configurationSetPositions := "Unit1.Em4.Config".cmAnodeMainPnP1AxisY.setPositions, moduleInterface := "Unit1.Em4.HmiInterface".cmAnodeMainPnP1AxisY, hmiInterface := "HMI_Interface_Parameter".TeachingPosInterface)
      "instTeachingPosAnodeMainPnP1AxisZ"(enable := "Unit1.EmNodes".unitStatus.mode.maintenance, selectTeachingPos := 12, indexTeachingPos := "HMI_Interface_Parameter".TeachingPosIndex, configurationSetPositions := "Unit1.Em4.Config".cmAnodeMainPnP1AxisZ.setPositions, moduleInterface := "Unit1.Em4.HmiInterface".cmAnodeMainPnP1AxisZ, hmiInterface := "HMI_Interface_Parameter".TeachingPosInterface)
   END_RUNG
   // the same network as SCL:
   "instTeachingPosCathodeMainPnP1AxisY"(enable := "Unit1.EmNodes".unitStatus.mode.maintenance,   // "LER_TeachingPos_Interface"
                           selectTeachingPos := 9,
                           indexTeachingPos := "HMI_Interface_Parameter".TeachingPosIndex,
                           configurationSetPositions := "Unit1.Em5.Config".cmCathodeMainPnP1AxisY.setPositions,
                           moduleInterface := "Unit1.Em5.HmiInterface".cmCathodeMainPnP1AxisY,
                           hmiInterface := "HMI_Interface_Parameter".TeachingPosInterface,
                           ENO => #_w1);
   "instTeachingPosCathodeMainPnP1AxisZ"(EN := #_w1,   // "LER_TeachingPos_Interface"
                           enable := "Unit1.EmNodes".unitStatus.mode.maintenance,
                           selectTeachingPos := 10,
                           indexTeachingPos := "HMI_Interface_Parameter".TeachingPosIndex,
                           configurationSetPositions := "Unit1.Em5.Config".cmCathodeMainPnP1AxisZ.setPositions,
                           moduleInterface := "Unit1.Em5.HmiInterface".cmCathodeMainPnP1AxisZ,
                           hmiInterface := "HMI_Interface_Parameter".TeachingPosInterface,
                           ENO => #_w2);
   "instTeachingPosAnodeMainPnP1AxisY"(EN := #_w2,   // "LER_TeachingPos_Interface"
                           enable := "Unit1.EmNodes".unitStatus.mode.maintenance,
                           selectTeachingPos := 11,
                           indexTeachingPos := "HMI_Interface_Parameter".TeachingPosIndex,
                           configurationSetPositions := "Unit1.Em4.Config".cmAnodeMainPnP1AxisY.setPositions,
                           moduleInterface := "Unit1.Em4.HmiInterface".cmAnodeMainPnP1AxisY,
                           hmiInterface := "HMI_Interface_Parameter".TeachingPosInterface,
                           ENO => #_w3);
   IF #_w3 THEN
       "instTeachingPosAnodeMainPnP1AxisZ"(enable := "Unit1.EmNodes".unitStatus.mode.maintenance,   // "LER_TeachingPos_Interface"
                               selectTeachingPos := 12,
                               indexTeachingPos := "HMI_Interface_Parameter".TeachingPosIndex,
                               configurationSetPositions := "Unit1.Em4.Config".cmAnodeMainPnP1AxisZ.setPositions,
                               moduleInterface := "Unit1.Em4.HmiInterface".cmAnodeMainPnP1AxisZ,
                               hmiInterface := "HMI_Interface_Parameter".TeachingPosInterface);
   END_IF;
END_REGION

REGION Network 20: Position Teaching (No 13~16)
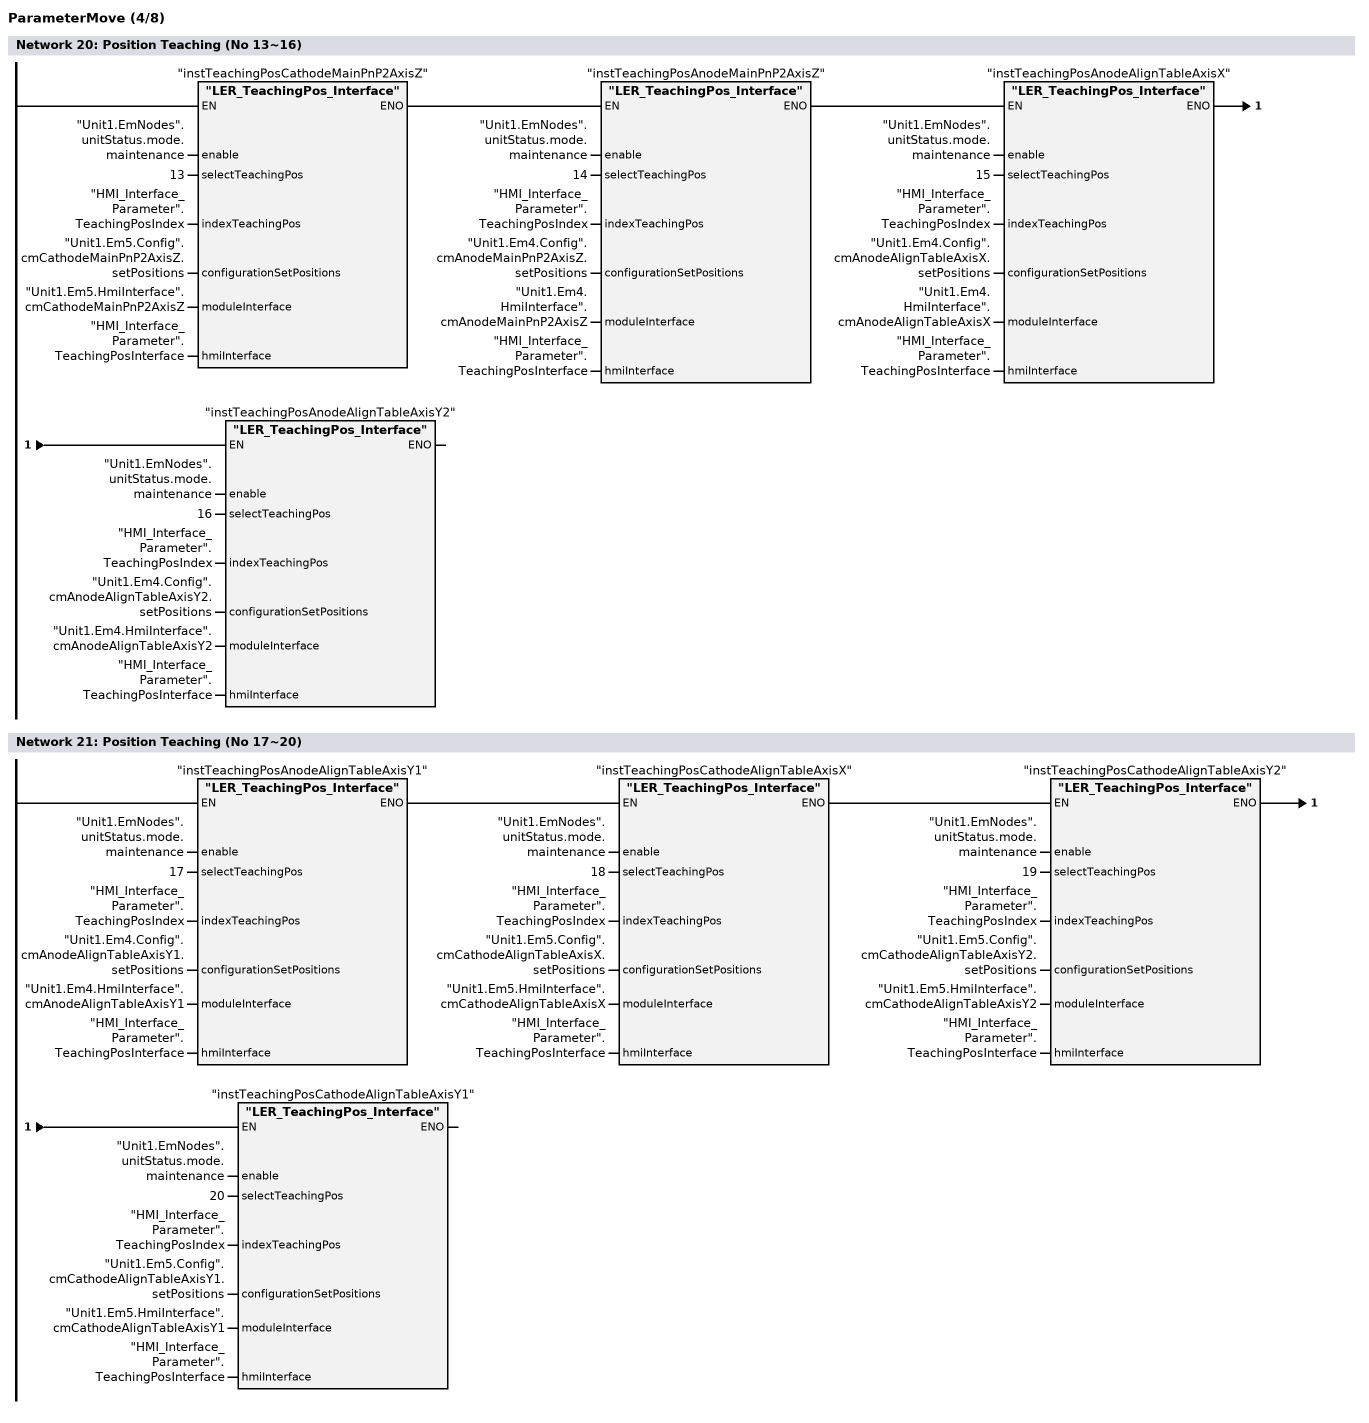
   RUNG wire#powerrail
      "instTeachingPosCathodeMainPnP2AxisZ"(enable := "Unit1.EmNodes".unitStatus.mode.maintenance, selectTeachingPos := 13, indexTeachingPos := "HMI_Interface_Parameter".TeachingPosIndex, configurationSetPositions := "Unit1.Em5.Config".cmCathodeMainPnP2AxisZ.setPositions, moduleInterface := "Unit1.Em5.HmiInterface".cmCathodeMainPnP2AxisZ, hmiInterface := "HMI_Interface_Parameter".TeachingPosInterface)
      "instTeachingPosAnodeMainPnP2AxisZ"(enable := "Unit1.EmNodes".unitStatus.mode.maintenance, selectTeachingPos := 14, indexTeachingPos := "HMI_Interface_Parameter".TeachingPosIndex, configurationSetPositions := "Unit1.Em4.Config".cmAnodeMainPnP2AxisZ.setPositions, moduleInterface := "Unit1.Em4.HmiInterface".cmAnodeMainPnP2AxisZ, hmiInterface := "HMI_Interface_Parameter".TeachingPosInterface)
      "instTeachingPosAnodeAlignTableAxisX"(enable := "Unit1.EmNodes".unitStatus.mode.maintenance, selectTeachingPos := 15, indexTeachingPos := "HMI_Interface_Parameter".TeachingPosIndex, configurationSetPositions := "Unit1.Em4.Config".cmAnodeAlignTableAxisX.setPositions, moduleInterface := "Unit1.Em4.HmiInterface".cmAnodeAlignTableAxisX, hmiInterface := "HMI_Interface_Parameter".TeachingPosInterface)
      "instTeachingPosAnodeAlignTableAxisY2"(enable := "Unit1.EmNodes".unitStatus.mode.maintenance, selectTeachingPos := 16, indexTeachingPos := "HMI_Interface_Parameter".TeachingPosIndex, configurationSetPositions := "Unit1.Em4.Config".cmAnodeAlignTableAxisY2.setPositions, moduleInterface := "Unit1.Em4.HmiInterface".cmAnodeAlignTableAxisY2, hmiInterface := "HMI_Interface_Parameter".TeachingPosInterface)
   END_RUNG
   // the same network as SCL:
   "instTeachingPosCathodeMainPnP2AxisZ"(enable := "Unit1.EmNodes".unitStatus.mode.maintenance,   // "LER_TeachingPos_Interface"
                           selectTeachingPos := 13,
                           indexTeachingPos := "HMI_Interface_Parameter".TeachingPosIndex,
                           configurationSetPositions := "Unit1.Em5.Config".cmCathodeMainPnP2AxisZ.setPositions,
                           moduleInterface := "Unit1.Em5.HmiInterface".cmCathodeMainPnP2AxisZ,
                           hmiInterface := "HMI_Interface_Parameter".TeachingPosInterface,
                           ENO => #_w1);
   "instTeachingPosAnodeMainPnP2AxisZ"(EN := #_w1,   // "LER_TeachingPos_Interface"
                           enable := "Unit1.EmNodes".unitStatus.mode.maintenance,
                           selectTeachingPos := 14,
                           indexTeachingPos := "HMI_Interface_Parameter".TeachingPosIndex,
                           configurationSetPositions := "Unit1.Em4.Config".cmAnodeMainPnP2AxisZ.setPositions,
                           moduleInterface := "Unit1.Em4.HmiInterface".cmAnodeMainPnP2AxisZ,
                           hmiInterface := "HMI_Interface_Parameter".TeachingPosInterface,
                           ENO => #_w2);
   "instTeachingPosAnodeAlignTableAxisX"(EN := #_w2,   // "LER_TeachingPos_Interface"
                           enable := "Unit1.EmNodes".unitStatus.mode.maintenance,
                           selectTeachingPos := 15,
                           indexTeachingPos := "HMI_Interface_Parameter".TeachingPosIndex,
                           configurationSetPositions := "Unit1.Em4.Config".cmAnodeAlignTableAxisX.setPositions,
                           moduleInterface := "Unit1.Em4.HmiInterface".cmAnodeAlignTableAxisX,
                           hmiInterface := "HMI_Interface_Parameter".TeachingPosInterface,
                           ENO => #_w3);
   IF #_w3 THEN
       "instTeachingPosAnodeAlignTableAxisY2"(enable := "Unit1.EmNodes".unitStatus.mode.maintenance,   // "LER_TeachingPos_Interface"
                               selectTeachingPos := 16,
                               indexTeachingPos := "HMI_Interface_Parameter".TeachingPosIndex,
                               configurationSetPositions := "Unit1.Em4.Config".cmAnodeAlignTableAxisY2.setPositions,
                               moduleInterface := "Unit1.Em4.HmiInterface".cmAnodeAlignTableAxisY2,
                               hmiInterface := "HMI_Interface_Parameter".TeachingPosInterface);
   END_IF;
END_REGION

REGION Network 21: Position Teaching (No 17~20)
   RUNG wire#powerrail
      "instTeachingPosAnodeAlignTableAxisY1"(enable := "Unit1.EmNodes".unitStatus.mode.maintenance, selectTeachingPos := 17, indexTeachingPos := "HMI_Interface_Parameter".TeachingPosIndex, configurationSetPositions := "Unit1.Em4.Config".cmAnodeAlignTableAxisY1.setPositions, moduleInterface := "Unit1.Em4.HmiInterface".cmAnodeAlignTableAxisY1, hmiInterface := "HMI_Interface_Parameter".TeachingPosInterface)
      "instTeachingPosCathodeAlignTableAxisX"(enable := "Unit1.EmNodes".unitStatus.mode.maintenance, selectTeachingPos := 18, indexTeachingPos := "HMI_Interface_Parameter".TeachingPosIndex, configurationSetPositions := "Unit1.Em5.Config".cmCathodeAlignTableAxisX.setPositions, moduleInterface := "Unit1.Em5.HmiInterface".cmCathodeAlignTableAxisX, hmiInterface := "HMI_Interface_Parameter".TeachingPosInterface)
      "instTeachingPosCathodeAlignTableAxisY2"(enable := "Unit1.EmNodes".unitStatus.mode.maintenance, selectTeachingPos := 19, indexTeachingPos := "HMI_Interface_Parameter".TeachingPosIndex, configurationSetPositions := "Unit1.Em5.Config".cmCathodeAlignTableAxisY2.setPositions, moduleInterface := "Unit1.Em5.HmiInterface".cmCathodeAlignTableAxisY2, hmiInterface := "HMI_Interface_Parameter".TeachingPosInterface)
      "instTeachingPosCathodeAlignTableAxisY1"(enable := "Unit1.EmNodes".unitStatus.mode.maintenance, selectTeachingPos := 20, indexTeachingPos := "HMI_Interface_Parameter".TeachingPosIndex, configurationSetPositions := "Unit1.Em5.Config".cmCathodeAlignTableAxisY1.setPositions, moduleInterface := "Unit1.Em5.HmiInterface".cmCathodeAlignTableAxisY1, hmiInterface := "HMI_Interface_Parameter".TeachingPosInterface)
   END_RUNG
   // the same network as SCL:
   "instTeachingPosAnodeAlignTableAxisY1"(enable := "Unit1.EmNodes".unitStatus.mode.maintenance,   // "LER_TeachingPos_Interface"
                           selectTeachingPos := 17,
                           indexTeachingPos := "HMI_Interface_Parameter".TeachingPosIndex,
                           configurationSetPositions := "Unit1.Em4.Config".cmAnodeAlignTableAxisY1.setPositions,
                           moduleInterface := "Unit1.Em4.HmiInterface".cmAnodeAlignTableAxisY1,
                           hmiInterface := "HMI_Interface_Parameter".TeachingPosInterface,
                           ENO => #_w1);
   "instTeachingPosCathodeAlignTableAxisX"(EN := #_w1,   // "LER_TeachingPos_Interface"
                           enable := "Unit1.EmNodes".unitStatus.mode.maintenance,
                           selectTeachingPos := 18,
                           indexTeachingPos := "HMI_Interface_Parameter".TeachingPosIndex,
                           configurationSetPositions := "Unit1.Em5.Config".cmCathodeAlignTableAxisX.setPositions,
                           moduleInterface := "Unit1.Em5.HmiInterface".cmCathodeAlignTableAxisX,
                           hmiInterface := "HMI_Interface_Parameter".TeachingPosInterface,
                           ENO => #_w2);
   "instTeachingPosCathodeAlignTableAxisY2"(EN := #_w2,   // "LER_TeachingPos_Interface"
                           enable := "Unit1.EmNodes".unitStatus.mode.maintenance,
                           selectTeachingPos := 19,
                           indexTeachingPos := "HMI_Interface_Parameter".TeachingPosIndex,
                           configurationSetPositions := "Unit1.Em5.Config".cmCathodeAlignTableAxisY2.setPositions,
                           moduleInterface := "Unit1.Em5.HmiInterface".cmCathodeAlignTableAxisY2,
                           hmiInterface := "HMI_Interface_Parameter".TeachingPosInterface,
                           ENO => #_w3);
   IF #_w3 THEN
       "instTeachingPosCathodeAlignTableAxisY1"(enable := "Unit1.EmNodes".unitStatus.mode.maintenance,   // "LER_TeachingPos_Interface"
                               selectTeachingPos := 20,
                               indexTeachingPos := "HMI_Interface_Parameter".TeachingPosIndex,
                               configurationSetPositions := "Unit1.Em5.Config".cmCathodeAlignTableAxisY1.setPositions,
                               moduleInterface := "Unit1.Em5.HmiInterface".cmCathodeAlignTableAxisY1,
                               hmiInterface := "HMI_Interface_Parameter".TeachingPosInterface);
   END_IF;
END_REGION

REGION Network 22: Position Teaching (No 21~24)
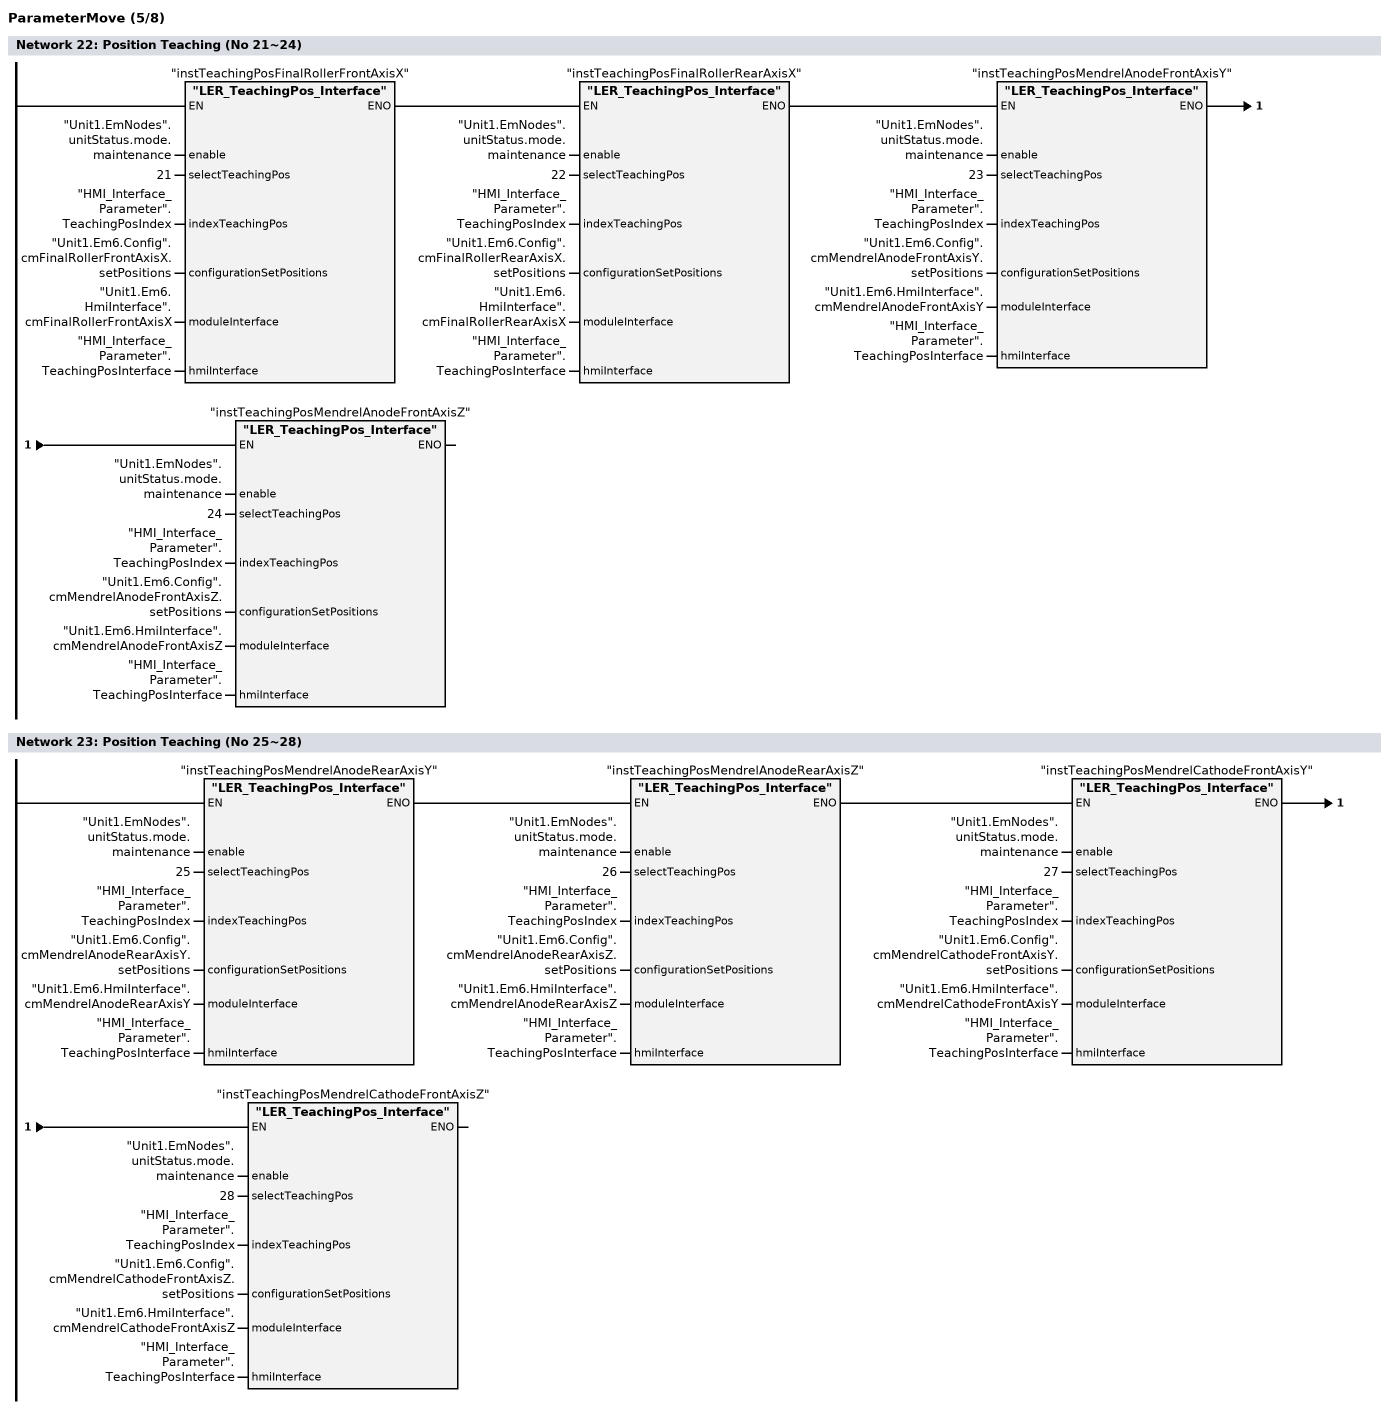
   RUNG wire#powerrail
      "instTeachingPosFinalRollerFrontAxisX"(enable := "Unit1.EmNodes".unitStatus.mode.maintenance, selectTeachingPos := 21, indexTeachingPos := "HMI_Interface_Parameter".TeachingPosIndex, configurationSetPositions := "Unit1.Em6.Config".cmFinalRollerFrontAxisX.setPositions, moduleInterface := "Unit1.Em6.HmiInterface".cmFinalRollerFrontAxisX, hmiInterface := "HMI_Interface_Parameter".TeachingPosInterface)
      "instTeachingPosFinalRollerRearAxisX"(enable := "Unit1.EmNodes".unitStatus.mode.maintenance, selectTeachingPos := 22, indexTeachingPos := "HMI_Interface_Parameter".TeachingPosIndex, configurationSetPositions := "Unit1.Em6.Config".cmFinalRollerRearAxisX.setPositions, moduleInterface := "Unit1.Em6.HmiInterface".cmFinalRollerRearAxisX, hmiInterface := "HMI_Interface_Parameter".TeachingPosInterface)
      "instTeachingPosMendrelAnodeFrontAxisY"(enable := "Unit1.EmNodes".unitStatus.mode.maintenance, selectTeachingPos := 23, indexTeachingPos := "HMI_Interface_Parameter".TeachingPosIndex, configurationSetPositions := "Unit1.Em6.Config".cmMendrelAnodeFrontAxisY.setPositions, moduleInterface := "Unit1.Em6.HmiInterface".cmMendrelAnodeFrontAxisY, hmiInterface := "HMI_Interface_Parameter".TeachingPosInterface)
      "instTeachingPosMendrelAnodeFrontAxisZ"(enable := "Unit1.EmNodes".unitStatus.mode.maintenance, selectTeachingPos := 24, indexTeachingPos := "HMI_Interface_Parameter".TeachingPosIndex, configurationSetPositions := "Unit1.Em6.Config".cmMendrelAnodeFrontAxisZ.setPositions, moduleInterface := "Unit1.Em6.HmiInterface".cmMendrelAnodeFrontAxisZ, hmiInterface := "HMI_Interface_Parameter".TeachingPosInterface)
   END_RUNG
   // the same network as SCL:
   "instTeachingPosFinalRollerFrontAxisX"(enable := "Unit1.EmNodes".unitStatus.mode.maintenance,   // "LER_TeachingPos_Interface"
                           selectTeachingPos := 21,
                           indexTeachingPos := "HMI_Interface_Parameter".TeachingPosIndex,
                           configurationSetPositions := "Unit1.Em6.Config".cmFinalRollerFrontAxisX.setPositions,
                           moduleInterface := "Unit1.Em6.HmiInterface".cmFinalRollerFrontAxisX,
                           hmiInterface := "HMI_Interface_Parameter".TeachingPosInterface,
                           ENO => #_w1);
   "instTeachingPosFinalRollerRearAxisX"(EN := #_w1,   // "LER_TeachingPos_Interface"
                           enable := "Unit1.EmNodes".unitStatus.mode.maintenance,
                           selectTeachingPos := 22,
                           indexTeachingPos := "HMI_Interface_Parameter".TeachingPosIndex,
                           configurationSetPositions := "Unit1.Em6.Config".cmFinalRollerRearAxisX.setPositions,
                           moduleInterface := "Unit1.Em6.HmiInterface".cmFinalRollerRearAxisX,
                           hmiInterface := "HMI_Interface_Parameter".TeachingPosInterface,
                           ENO => #_w2);
   "instTeachingPosMendrelAnodeFrontAxisY"(EN := #_w2,   // "LER_TeachingPos_Interface"
                           enable := "Unit1.EmNodes".unitStatus.mode.maintenance,
                           selectTeachingPos := 23,
                           indexTeachingPos := "HMI_Interface_Parameter".TeachingPosIndex,
                           configurationSetPositions := "Unit1.Em6.Config".cmMendrelAnodeFrontAxisY.setPositions,
                           moduleInterface := "Unit1.Em6.HmiInterface".cmMendrelAnodeFrontAxisY,
                           hmiInterface := "HMI_Interface_Parameter".TeachingPosInterface,
                           ENO => #_w3);
   IF #_w3 THEN
       "instTeachingPosMendrelAnodeFrontAxisZ"(enable := "Unit1.EmNodes".unitStatus.mode.maintenance,   // "LER_TeachingPos_Interface"
                               selectTeachingPos := 24,
                               indexTeachingPos := "HMI_Interface_Parameter".TeachingPosIndex,
                               configurationSetPositions := "Unit1.Em6.Config".cmMendrelAnodeFrontAxisZ.setPositions,
                               moduleInterface := "Unit1.Em6.HmiInterface".cmMendrelAnodeFrontAxisZ,
                               hmiInterface := "HMI_Interface_Parameter".TeachingPosInterface);
   END_IF;
END_REGION

REGION Network 23: Position Teaching (No 25~28)
   RUNG wire#powerrail
      "instTeachingPosMendrelAnodeRearAxisY"(enable := "Unit1.EmNodes".unitStatus.mode.maintenance, selectTeachingPos := 25, indexTeachingPos := "HMI_Interface_Parameter".TeachingPosIndex, configurationSetPositions := "Unit1.Em6.Config".cmMendrelAnodeRearAxisY.setPositions, moduleInterface := "Unit1.Em6.HmiInterface".cmMendrelAnodeRearAxisY, hmiInterface := "HMI_Interface_Parameter".TeachingPosInterface)
      "instTeachingPosMendrelAnodeRearAxisZ"(enable := "Unit1.EmNodes".unitStatus.mode.maintenance, selectTeachingPos := 26, indexTeachingPos := "HMI_Interface_Parameter".TeachingPosIndex, configurationSetPositions := "Unit1.Em6.Config".cmMendrelAnodeRearAxisZ.setPositions, moduleInterface := "Unit1.Em6.HmiInterface".cmMendrelAnodeRearAxisZ, hmiInterface := "HMI_Interface_Parameter".TeachingPosInterface)
      "instTeachingPosMendrelCathodeFrontAxisY"(enable := "Unit1.EmNodes".unitStatus.mode.maintenance, selectTeachingPos := 27, indexTeachingPos := "HMI_Interface_Parameter".TeachingPosIndex, configurationSetPositions := "Unit1.Em6.Config".cmMendrelCathodeFrontAxisY.setPositions, moduleInterface := "Unit1.Em6.HmiInterface".cmMendrelCathodeFrontAxisY, hmiInterface := "HMI_Interface_Parameter".TeachingPosInterface)
      "instTeachingPosMendrelCathodeFrontAxisZ"(enable := "Unit1.EmNodes".unitStatus.mode.maintenance, selectTeachingPos := 28, indexTeachingPos := "HMI_Interface_Parameter".TeachingPosIndex, configurationSetPositions := "Unit1.Em6.Config".cmMendrelCathodeFrontAxisZ.setPositions, moduleInterface := "Unit1.Em6.HmiInterface".cmMendrelCathodeFrontAxisZ, hmiInterface := "HMI_Interface_Parameter".TeachingPosInterface)
   END_RUNG
   // the same network as SCL:
   "instTeachingPosMendrelAnodeRearAxisY"(enable := "Unit1.EmNodes".unitStatus.mode.maintenance,   // "LER_TeachingPos_Interface"
                           selectTeachingPos := 25,
                           indexTeachingPos := "HMI_Interface_Parameter".TeachingPosIndex,
                           configurationSetPositions := "Unit1.Em6.Config".cmMendrelAnodeRearAxisY.setPositions,
                           moduleInterface := "Unit1.Em6.HmiInterface".cmMendrelAnodeRearAxisY,
                           hmiInterface := "HMI_Interface_Parameter".TeachingPosInterface,
                           ENO => #_w1);
   "instTeachingPosMendrelAnodeRearAxisZ"(EN := #_w1,   // "LER_TeachingPos_Interface"
                           enable := "Unit1.EmNodes".unitStatus.mode.maintenance,
                           selectTeachingPos := 26,
                           indexTeachingPos := "HMI_Interface_Parameter".TeachingPosIndex,
                           configurationSetPositions := "Unit1.Em6.Config".cmMendrelAnodeRearAxisZ.setPositions,
                           moduleInterface := "Unit1.Em6.HmiInterface".cmMendrelAnodeRearAxisZ,
                           hmiInterface := "HMI_Interface_Parameter".TeachingPosInterface,
                           ENO => #_w2);
   "instTeachingPosMendrelCathodeFrontAxisY"(EN := #_w2,   // "LER_TeachingPos_Interface"
                           enable := "Unit1.EmNodes".unitStatus.mode.maintenance,
                           selectTeachingPos := 27,
                           indexTeachingPos := "HMI_Interface_Parameter".TeachingPosIndex,
                           configurationSetPositions := "Unit1.Em6.Config".cmMendrelCathodeFrontAxisY.setPositions,
                           moduleInterface := "Unit1.Em6.HmiInterface".cmMendrelCathodeFrontAxisY,
                           hmiInterface := "HMI_Interface_Parameter".TeachingPosInterface,
                           ENO => #_w3);
   IF #_w3 THEN
       "instTeachingPosMendrelCathodeFrontAxisZ"(enable := "Unit1.EmNodes".unitStatus.mode.maintenance,   // "LER_TeachingPos_Interface"
                               selectTeachingPos := 28,
                               indexTeachingPos := "HMI_Interface_Parameter".TeachingPosIndex,
                               configurationSetPositions := "Unit1.Em6.Config".cmMendrelCathodeFrontAxisZ.setPositions,
                               moduleInterface := "Unit1.Em6.HmiInterface".cmMendrelCathodeFrontAxisZ,
                               hmiInterface := "HMI_Interface_Parameter".TeachingPosInterface);
   END_IF;
END_REGION

REGION Network 24: Position Teaching (No 29~32)
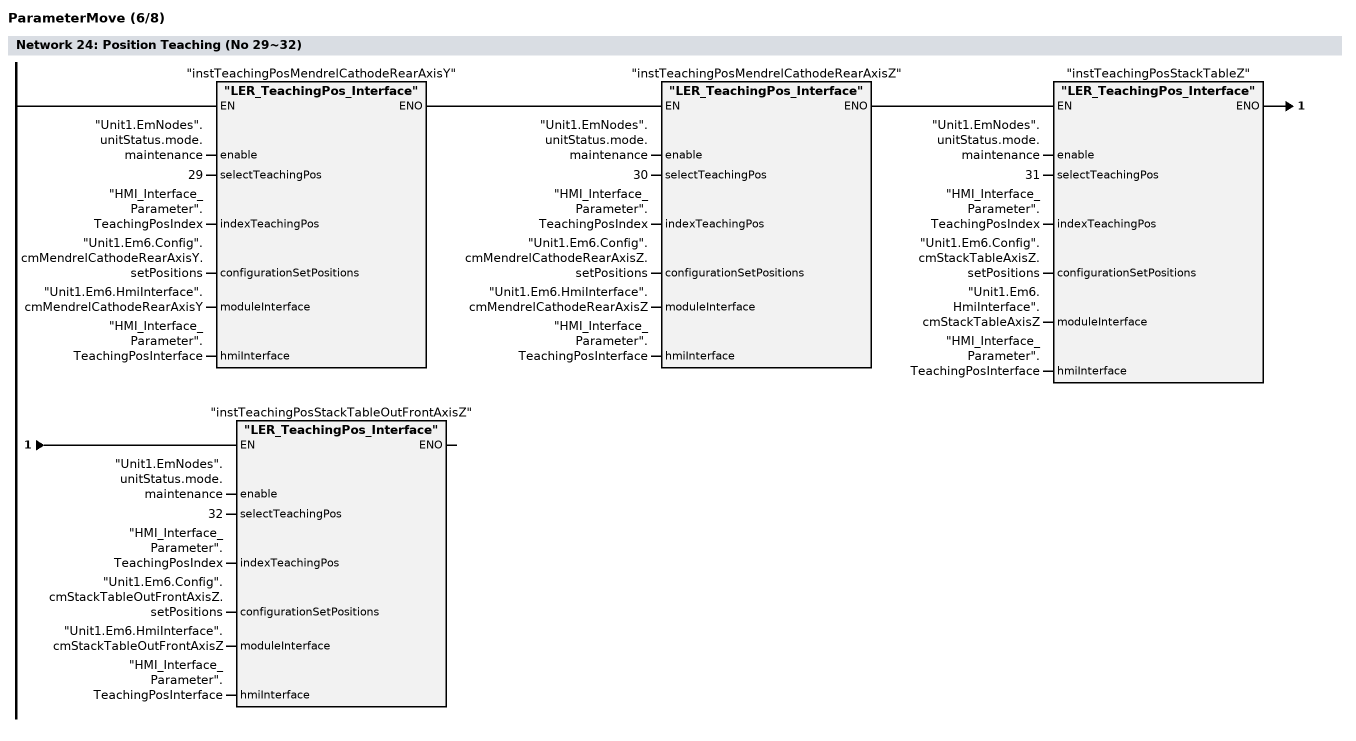
   RUNG wire#powerrail
      "instTeachingPosMendrelCathodeRearAxisY"(enable := "Unit1.EmNodes".unitStatus.mode.maintenance, selectTeachingPos := 29, indexTeachingPos := "HMI_Interface_Parameter".TeachingPosIndex, configurationSetPositions := "Unit1.Em6.Config".cmMendrelCathodeRearAxisY.setPositions, moduleInterface := "Unit1.Em6.HmiInterface".cmMendrelCathodeRearAxisY, hmiInterface := "HMI_Interface_Parameter".TeachingPosInterface)
      "instTeachingPosMendrelCathodeRearAxisZ"(enable := "Unit1.EmNodes".unitStatus.mode.maintenance, selectTeachingPos := 30, indexTeachingPos := "HMI_Interface_Parameter".TeachingPosIndex, configurationSetPositions := "Unit1.Em6.Config".cmMendrelCathodeRearAxisZ.setPositions, moduleInterface := "Unit1.Em6.HmiInterface".cmMendrelCathodeRearAxisZ, hmiInterface := "HMI_Interface_Parameter".TeachingPosInterface)
      "instTeachingPosStackTableZ"(enable := "Unit1.EmNodes".unitStatus.mode.maintenance, selectTeachingPos := 31, indexTeachingPos := "HMI_Interface_Parameter".TeachingPosIndex, configurationSetPositions := "Unit1.Em6.Config".cmStackTableAxisZ.setPositions, moduleInterface := "Unit1.Em6.HmiInterface".cmStackTableAxisZ, hmiInterface := "HMI_Interface_Parameter".TeachingPosInterface)
      "instTeachingPosStackTableOutFrontAxisZ"(enable := "Unit1.EmNodes".unitStatus.mode.maintenance, selectTeachingPos := 32, indexTeachingPos := "HMI_Interface_Parameter".TeachingPosIndex, configurationSetPositions := "Unit1.Em6.Config".cmStackTableOutFrontAxisZ.setPositions, moduleInterface := "Unit1.Em6.HmiInterface".cmStackTableOutFrontAxisZ, hmiInterface := "HMI_Interface_Parameter".TeachingPosInterface)
   END_RUNG
   // the same network as SCL:
   "instTeachingPosMendrelCathodeRearAxisY"(enable := "Unit1.EmNodes".unitStatus.mode.maintenance,   // "LER_TeachingPos_Interface"
                           selectTeachingPos := 29,
                           indexTeachingPos := "HMI_Interface_Parameter".TeachingPosIndex,
                           configurationSetPositions := "Unit1.Em6.Config".cmMendrelCathodeRearAxisY.setPositions,
                           moduleInterface := "Unit1.Em6.HmiInterface".cmMendrelCathodeRearAxisY,
                           hmiInterface := "HMI_Interface_Parameter".TeachingPosInterface,
                           ENO => #_w1);
   "instTeachingPosMendrelCathodeRearAxisZ"(EN := #_w1,   // "LER_TeachingPos_Interface"
                           enable := "Unit1.EmNodes".unitStatus.mode.maintenance,
                           selectTeachingPos := 30,
                           indexTeachingPos := "HMI_Interface_Parameter".TeachingPosIndex,
                           configurationSetPositions := "Unit1.Em6.Config".cmMendrelCathodeRearAxisZ.setPositions,
                           moduleInterface := "Unit1.Em6.HmiInterface".cmMendrelCathodeRearAxisZ,
                           hmiInterface := "HMI_Interface_Parameter".TeachingPosInterface,
                           ENO => #_w2);
   "instTeachingPosStackTableZ"(EN := #_w2,   // "LER_TeachingPos_Interface"
                           enable := "Unit1.EmNodes".unitStatus.mode.maintenance,
                           selectTeachingPos := 31,
                           indexTeachingPos := "HMI_Interface_Parameter".TeachingPosIndex,
                           configurationSetPositions := "Unit1.Em6.Config".cmStackTableAxisZ.setPositions,
                           moduleInterface := "Unit1.Em6.HmiInterface".cmStackTableAxisZ,
                           hmiInterface := "HMI_Interface_Parameter".TeachingPosInterface,
                           ENO => #_w3);
   IF #_w3 THEN
       "instTeachingPosStackTableOutFrontAxisZ"(enable := "Unit1.EmNodes".unitStatus.mode.maintenance,   // "LER_TeachingPos_Interface"
                               selectTeachingPos := 32,
                               indexTeachingPos := "HMI_Interface_Parameter".TeachingPosIndex,
                               configurationSetPositions := "Unit1.Em6.Config".cmStackTableOutFrontAxisZ.setPositions,
                               moduleInterface := "Unit1.Em6.HmiInterface".cmStackTableOutFrontAxisZ,
                               hmiInterface := "HMI_Interface_Parameter".TeachingPosInterface);
   END_IF;
END_REGION

REGION Network 25: Position Teaching (No 33~36)
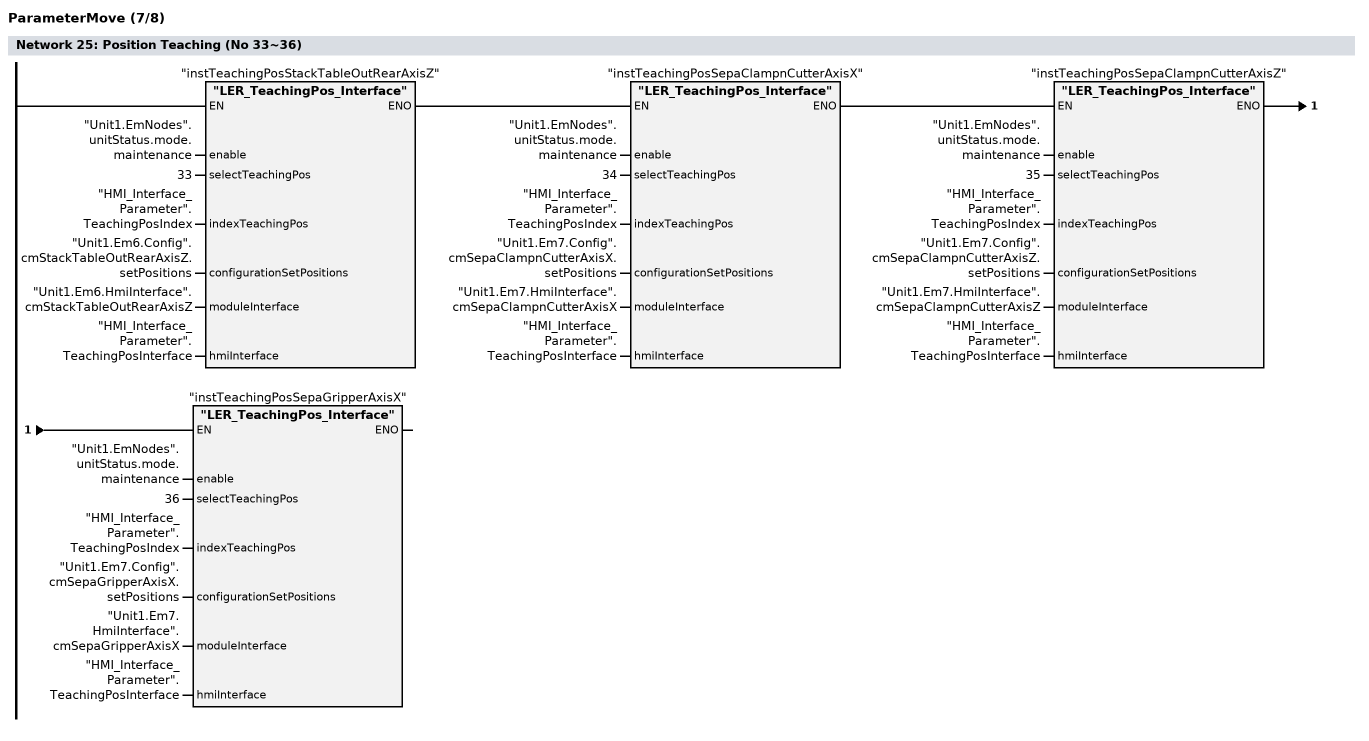
   RUNG wire#powerrail
      "instTeachingPosStackTableOutRearAxisZ"(enable := "Unit1.EmNodes".unitStatus.mode.maintenance, selectTeachingPos := 33, indexTeachingPos := "HMI_Interface_Parameter".TeachingPosIndex, configurationSetPositions := "Unit1.Em6.Config".cmStackTableOutRearAxisZ.setPositions, moduleInterface := "Unit1.Em6.HmiInterface".cmStackTableOutRearAxisZ, hmiInterface := "HMI_Interface_Parameter".TeachingPosInterface)
      "instTeachingPosSepaClampnCutterAxisX"(enable := "Unit1.EmNodes".unitStatus.mode.maintenance, selectTeachingPos := 34, indexTeachingPos := "HMI_Interface_Parameter".TeachingPosIndex, configurationSetPositions := "Unit1.Em7.Config".cmSepaClampnCutterAxisX.setPositions, moduleInterface := "Unit1.Em7.HmiInterface".cmSepaClampnCutterAxisX, hmiInterface := "HMI_Interface_Parameter".TeachingPosInterface)
      "instTeachingPosSepaClampnCutterAxisZ"(enable := "Unit1.EmNodes".unitStatus.mode.maintenance, selectTeachingPos := 35, indexTeachingPos := "HMI_Interface_Parameter".TeachingPosIndex, configurationSetPositions := "Unit1.Em7.Config".cmSepaClampnCutterAxisZ.setPositions, moduleInterface := "Unit1.Em7.HmiInterface".cmSepaClampnCutterAxisZ, hmiInterface := "HMI_Interface_Parameter".TeachingPosInterface)
      "instTeachingPosSepaGripperAxisX"(enable := "Unit1.EmNodes".unitStatus.mode.maintenance, selectTeachingPos := 36, indexTeachingPos := "HMI_Interface_Parameter".TeachingPosIndex, configurationSetPositions := "Unit1.Em7.Config".cmSepaGripperAxisX.setPositions, moduleInterface := "Unit1.Em7.HmiInterface".cmSepaGripperAxisX, hmiInterface := "HMI_Interface_Parameter".TeachingPosInterface)
   END_RUNG
   // the same network as SCL:
   "instTeachingPosStackTableOutRearAxisZ"(enable := "Unit1.EmNodes".unitStatus.mode.maintenance,   // "LER_TeachingPos_Interface"
                           selectTeachingPos := 33,
                           indexTeachingPos := "HMI_Interface_Parameter".TeachingPosIndex,
                           configurationSetPositions := "Unit1.Em6.Config".cmStackTableOutRearAxisZ.setPositions,
                           moduleInterface := "Unit1.Em6.HmiInterface".cmStackTableOutRearAxisZ,
                           hmiInterface := "HMI_Interface_Parameter".TeachingPosInterface,
                           ENO => #_w1);
   "instTeachingPosSepaClampnCutterAxisX"(EN := #_w1,   // "LER_TeachingPos_Interface"
                           enable := "Unit1.EmNodes".unitStatus.mode.maintenance,
                           selectTeachingPos := 34,
                           indexTeachingPos := "HMI_Interface_Parameter".TeachingPosIndex,
                           configurationSetPositions := "Unit1.Em7.Config".cmSepaClampnCutterAxisX.setPositions,
                           moduleInterface := "Unit1.Em7.HmiInterface".cmSepaClampnCutterAxisX,
                           hmiInterface := "HMI_Interface_Parameter".TeachingPosInterface,
                           ENO => #_w2);
   "instTeachingPosSepaClampnCutterAxisZ"(EN := #_w2,   // "LER_TeachingPos_Interface"
                           enable := "Unit1.EmNodes".unitStatus.mode.maintenance,
                           selectTeachingPos := 35,
                           indexTeachingPos := "HMI_Interface_Parameter".TeachingPosIndex,
                           configurationSetPositions := "Unit1.Em7.Config".cmSepaClampnCutterAxisZ.setPositions,
                           moduleInterface := "Unit1.Em7.HmiInterface".cmSepaClampnCutterAxisZ,
                           hmiInterface := "HMI_Interface_Parameter".TeachingPosInterface,
                           ENO => #_w3);
   IF #_w3 THEN
       "instTeachingPosSepaGripperAxisX"(enable := "Unit1.EmNodes".unitStatus.mode.maintenance,   // "LER_TeachingPos_Interface"
                               selectTeachingPos := 36,
                               indexTeachingPos := "HMI_Interface_Parameter".TeachingPosIndex,
                               configurationSetPositions := "Unit1.Em7.Config".cmSepaGripperAxisX.setPositions,
                               moduleInterface := "Unit1.Em7.HmiInterface".cmSepaGripperAxisX,
                               hmiInterface := "HMI_Interface_Parameter".TeachingPosInterface);
   END_IF;
END_REGION

REGION Network 26: Position Teaching (No 37~40)
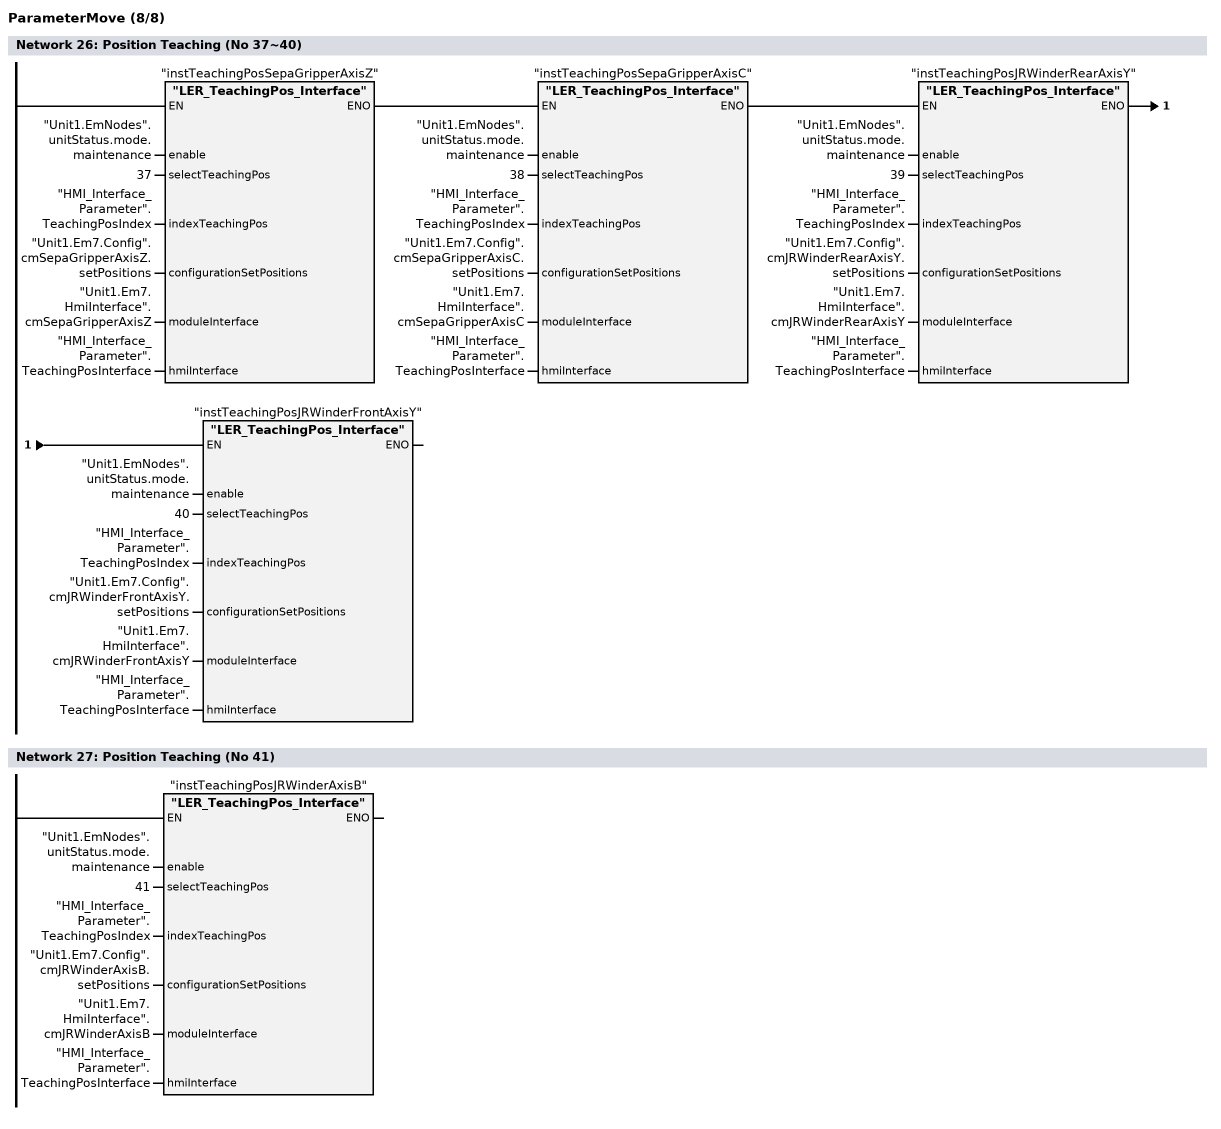
   RUNG wire#powerrail
      "instTeachingPosSepaGripperAxisZ"(enable := "Unit1.EmNodes".unitStatus.mode.maintenance, selectTeachingPos := 37, indexTeachingPos := "HMI_Interface_Parameter".TeachingPosIndex, configurationSetPositions := "Unit1.Em7.Config".cmSepaGripperAxisZ.setPositions, moduleInterface := "Unit1.Em7.HmiInterface".cmSepaGripperAxisZ, hmiInterface := "HMI_Interface_Parameter".TeachingPosInterface)
      "instTeachingPosSepaGripperAxisC"(enable := "Unit1.EmNodes".unitStatus.mode.maintenance, selectTeachingPos := 38, indexTeachingPos := "HMI_Interface_Parameter".TeachingPosIndex, configurationSetPositions := "Unit1.Em7.Config".cmSepaGripperAxisC.setPositions, moduleInterface := "Unit1.Em7.HmiInterface".cmSepaGripperAxisC, hmiInterface := "HMI_Interface_Parameter".TeachingPosInterface)
      "instTeachingPosJRWinderRearAxisY"(enable := "Unit1.EmNodes".unitStatus.mode.maintenance, selectTeachingPos := 39, indexTeachingPos := "HMI_Interface_Parameter".TeachingPosIndex, configurationSetPositions := "Unit1.Em7.Config".cmJRWinderRearAxisY.setPositions, moduleInterface := "Unit1.Em7.HmiInterface".cmJRWinderRearAxisY, hmiInterface := "HMI_Interface_Parameter".TeachingPosInterface)
      "instTeachingPosJRWinderFrontAxisY"(enable := "Unit1.EmNodes".unitStatus.mode.maintenance, selectTeachingPos := 40, indexTeachingPos := "HMI_Interface_Parameter".TeachingPosIndex, configurationSetPositions := "Unit1.Em7.Config".cmJRWinderFrontAxisY.setPositions, moduleInterface := "Unit1.Em7.HmiInterface".cmJRWinderFrontAxisY, hmiInterface := "HMI_Interface_Parameter".TeachingPosInterface)
   END_RUNG
   // the same network as SCL:
   "instTeachingPosSepaGripperAxisZ"(enable := "Unit1.EmNodes".unitStatus.mode.maintenance,   // "LER_TeachingPos_Interface"
                           selectTeachingPos := 37,
                           indexTeachingPos := "HMI_Interface_Parameter".TeachingPosIndex,
                           configurationSetPositions := "Unit1.Em7.Config".cmSepaGripperAxisZ.setPositions,
                           moduleInterface := "Unit1.Em7.HmiInterface".cmSepaGripperAxisZ,
                           hmiInterface := "HMI_Interface_Parameter".TeachingPosInterface,
                           ENO => #_w1);
   "instTeachingPosSepaGripperAxisC"(EN := #_w1,   // "LER_TeachingPos_Interface"
                           enable := "Unit1.EmNodes".unitStatus.mode.maintenance,
                           selectTeachingPos := 38,
                           indexTeachingPos := "HMI_Interface_Parameter".TeachingPosIndex,
                           configurationSetPositions := "Unit1.Em7.Config".cmSepaGripperAxisC.setPositions,
                           moduleInterface := "Unit1.Em7.HmiInterface".cmSepaGripperAxisC,
                           hmiInterface := "HMI_Interface_Parameter".TeachingPosInterface,
                           ENO => #_w2);
   "instTeachingPosJRWinderRearAxisY"(EN := #_w2,   // "LER_TeachingPos_Interface"
                           enable := "Unit1.EmNodes".unitStatus.mode.maintenance,
                           selectTeachingPos := 39,
                           indexTeachingPos := "HMI_Interface_Parameter".TeachingPosIndex,
                           configurationSetPositions := "Unit1.Em7.Config".cmJRWinderRearAxisY.setPositions,
                           moduleInterface := "Unit1.Em7.HmiInterface".cmJRWinderRearAxisY,
                           hmiInterface := "HMI_Interface_Parameter".TeachingPosInterface,
                           ENO => #_w3);
   IF #_w3 THEN
       "instTeachingPosJRWinderFrontAxisY"(enable := "Unit1.EmNodes".unitStatus.mode.maintenance,   // "LER_TeachingPos_Interface"
                               selectTeachingPos := 40,
                               indexTeachingPos := "HMI_Interface_Parameter".TeachingPosIndex,
                               configurationSetPositions := "Unit1.Em7.Config".cmJRWinderFrontAxisY.setPositions,
                               moduleInterface := "Unit1.Em7.HmiInterface".cmJRWinderFrontAxisY,
                               hmiInterface := "HMI_Interface_Parameter".TeachingPosInterface);
   END_IF;
END_REGION

REGION Network 27: Position Teaching (No 41)
   RUNG wire#powerrail
      "instTeachingPosJRWinderAxisB"(enable := "Unit1.EmNodes".unitStatus.mode.maintenance, selectTeachingPos := 41, indexTeachingPos := "HMI_Interface_Parameter".TeachingPosIndex, configurationSetPositions := "Unit1.Em7.Config".cmJRWinderAxisB.setPositions, moduleInterface := "Unit1.Em7.HmiInterface".cmJRWinderAxisB, hmiInterface := "HMI_Interface_Parameter".TeachingPosInterface)
   END_RUNG
   // the same network as SCL:
   "instTeachingPosJRWinderAxisB"(enable := "Unit1.EmNodes".unitStatus.mode.maintenance,   // "LER_TeachingPos_Interface"
                           selectTeachingPos := 41,
                           indexTeachingPos := "HMI_Interface_Parameter".TeachingPosIndex,
                           configurationSetPositions := "Unit1.Em7.Config".cmJRWinderAxisB.setPositions,
                           moduleInterface := "Unit1.Em7.HmiInterface".cmJRWinderAxisB,
                           hmiInterface := "HMI_Interface_Parameter".TeachingPosInterface);
END_REGION
END_FUNCTION

FUNCTION "CallManualOperationLines_Unit1" : Void   // FC83, LAD
// stored: SetENOAutomatically false
   VAR_TEMP
      StatusEm : Array[0..7] of Struct
         Status : Array[0..40] of Word;
      END_STRUCT;
      errorIDEm : Array[0..7] of Struct
         errorID : Array[0..40] of Word;
      END_STRUCT;
      disableUnit1 : Bool;
      TempAxisCommands : "LBC_typeAxis64PosManualCommands";
      TempAxisMonitoring : "LBC_typeAxis64PosProcessValues";
      TempSoftCam : Array[0..8] of "LER_typeSoftCamParameter";
   END_VAR
   VAR CONSTANT
      MECHANIC_NAME_ENABLE : Bool;
   END_VAR
   VAR_TEMP   // added for the SCL form of the ladder/FBD networks
      _w1 : Bool;
   END_VAR
BEGIN

REGION Network 1: Unit 1 Enable Manual Operation
   // Condition to disable manual operation lines in Unit 3
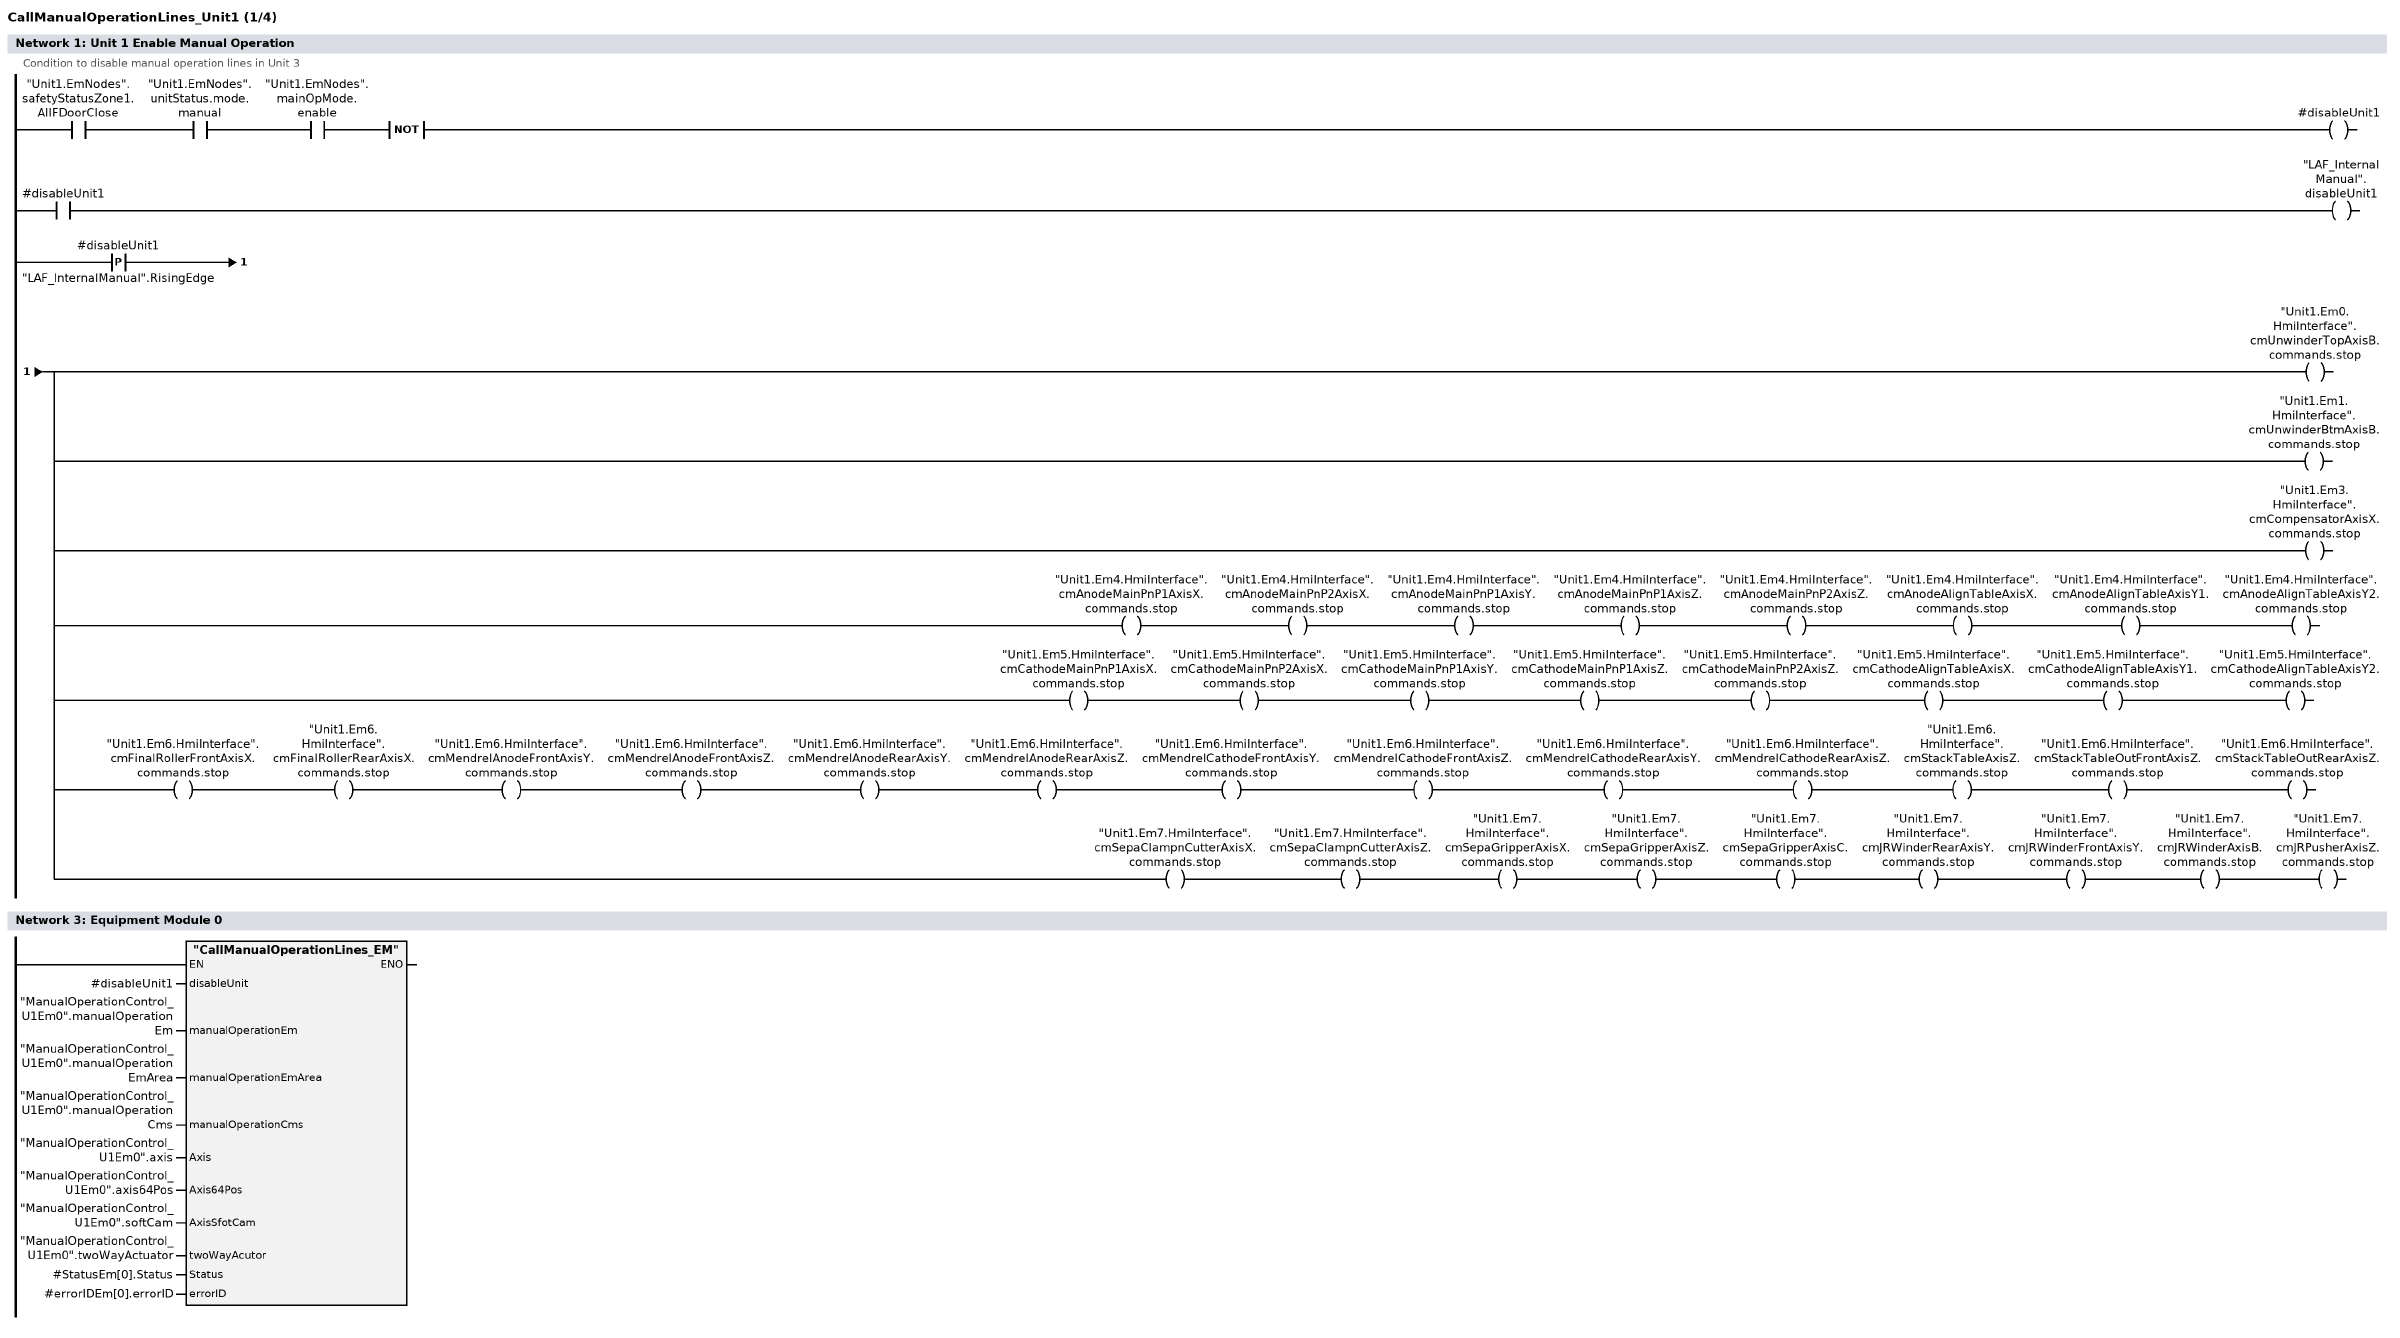
   RUNG wire#powerrail
      Contact( "Unit1.EmNodes".safetyStatusZone1.AllFDoorClose )
      Contact( "Unit1.EmNodes".unitStatus.mode.manual )
      Contact( "Unit1.EmNodes".mainOpMode.enable )
      Not()
      Coil( #disableUnit1 )
   END_RUNG
   RUNG wire#powerrail
      Contact( #disableUnit1 )
      Coil( "LAF_InternalManual".disableUnit1 )
   END_RUNG
   RUNG wire#powerrail
      P_Contact(operand := #disableUnit1, bit := "LAF_InternalManual".RisingEdge)
      wire#w1
      Coil( "Unit1.Em0.HmiInterface".cmUnwinderTopAxisB.commands.stop )
   END_RUNG
   RUNG wire#w1
      Coil( "Unit1.Em1.HmiInterface".cmUnwinderBtmAxisB.commands.stop )
   END_RUNG
   RUNG wire#w1
      Coil( "Unit1.Em3.HmiInterface".cmCompensatorAxisX.commands.stop )
   END_RUNG
   RUNG wire#w1
      Coil( "Unit1.Em4.HmiInterface".cmAnodeMainPnP1AxisX.commands.stop )
      Coil( "Unit1.Em4.HmiInterface".cmAnodeMainPnP2AxisX.commands.stop )
      Coil( "Unit1.Em4.HmiInterface".cmAnodeMainPnP1AxisY.commands.stop )
      Coil( "Unit1.Em4.HmiInterface".cmAnodeMainPnP1AxisZ.commands.stop )
      Coil( "Unit1.Em4.HmiInterface".cmAnodeMainPnP2AxisZ.commands.stop )
      Coil( "Unit1.Em4.HmiInterface".cmAnodeAlignTableAxisX.commands.stop )
      Coil( "Unit1.Em4.HmiInterface".cmAnodeAlignTableAxisY1.commands.stop )
      Coil( "Unit1.Em4.HmiInterface".cmAnodeAlignTableAxisY2.commands.stop )
   END_RUNG
   RUNG wire#w1
      Coil( "Unit1.Em5.HmiInterface".cmCathodeMainPnP1AxisX.commands.stop )
      Coil( "Unit1.Em5.HmiInterface".cmCathodeMainPnP2AxisX.commands.stop )
      Coil( "Unit1.Em5.HmiInterface".cmCathodeMainPnP1AxisY.commands.stop )
      Coil( "Unit1.Em5.HmiInterface".cmCathodeMainPnP1AxisZ.commands.stop )
      Coil( "Unit1.Em5.HmiInterface".cmCathodeMainPnP2AxisZ.commands.stop )
      Coil( "Unit1.Em5.HmiInterface".cmCathodeAlignTableAxisX.commands.stop )
      Coil( "Unit1.Em5.HmiInterface".cmCathodeAlignTableAxisY1.commands.stop )
      Coil( "Unit1.Em5.HmiInterface".cmCathodeAlignTableAxisY2.commands.stop )
   END_RUNG
   RUNG wire#w1
      Coil( "Unit1.Em6.HmiInterface".cmFinalRollerFrontAxisX.commands.stop )
      Coil( "Unit1.Em6.HmiInterface".cmFinalRollerRearAxisX.commands.stop )
      Coil( "Unit1.Em6.HmiInterface".cmMendrelAnodeFrontAxisY.commands.stop )
      Coil( "Unit1.Em6.HmiInterface".cmMendrelAnodeFrontAxisZ.commands.stop )
      Coil( "Unit1.Em6.HmiInterface".cmMendrelAnodeRearAxisY.commands.stop )
      Coil( "Unit1.Em6.HmiInterface".cmMendrelAnodeRearAxisZ.commands.stop )
      Coil( "Unit1.Em6.HmiInterface".cmMendrelCathodeFrontAxisY.commands.stop )
      Coil( "Unit1.Em6.HmiInterface".cmMendrelCathodeFrontAxisZ.commands.stop )
      Coil( "Unit1.Em6.HmiInterface".cmMendrelCathodeRearAxisY.commands.stop )
      Coil( "Unit1.Em6.HmiInterface".cmMendrelCathodeRearAxisZ.commands.stop )
      Coil( "Unit1.Em6.HmiInterface".cmStackTableAxisZ.commands.stop )
      Coil( "Unit1.Em6.HmiInterface".cmStackTableOutFrontAxisZ.commands.stop )
      Coil( "Unit1.Em6.HmiInterface".cmStackTableOutRearAxisZ.commands.stop )
   END_RUNG
   RUNG wire#w1
      Coil( "Unit1.Em7.HmiInterface".cmSepaClampnCutterAxisX.commands.stop )
      Coil( "Unit1.Em7.HmiInterface".cmSepaClampnCutterAxisZ.commands.stop )
      Coil( "Unit1.Em7.HmiInterface".cmSepaGripperAxisX.commands.stop )
      Coil( "Unit1.Em7.HmiInterface".cmSepaGripperAxisZ.commands.stop )
      Coil( "Unit1.Em7.HmiInterface".cmSepaGripperAxisC.commands.stop )
      Coil( "Unit1.Em7.HmiInterface".cmJRWinderRearAxisY.commands.stop )
      Coil( "Unit1.Em7.HmiInterface".cmJRWinderFrontAxisY.commands.stop )
      Coil( "Unit1.Em7.HmiInterface".cmJRWinderAxisB.commands.stop )
      Coil( "Unit1.Em7.HmiInterface".cmJRPusherAxisZ.commands.stop )
   END_RUNG
   // the same network as SCL:
   #disableUnit1 := NOT ("Unit1.EmNodes".safetyStatusZone1.AllFDoorClose AND "Unit1.EmNodes".unitStatus.mode.manual AND "Unit1.EmNodes".mainOpMode.enable);
   "LAF_InternalManual".disableUnit1 := #disableUnit1;
   #_w1 := #disableUnit1 AND NOT "LAF_InternalManual".RisingEdge;   // rising edge of #disableUnit1
   "LAF_InternalManual".RisingEdge := #disableUnit1;
   "Unit1.Em0.HmiInterface".cmUnwinderTopAxisB.commands.stop := #_w1;
   "Unit1.Em1.HmiInterface".cmUnwinderBtmAxisB.commands.stop := #_w1;
   "Unit1.Em3.HmiInterface".cmCompensatorAxisX.commands.stop := #_w1;
   "Unit1.Em4.HmiInterface".cmAnodeMainPnP1AxisX.commands.stop := #_w1;
   "Unit1.Em4.HmiInterface".cmAnodeMainPnP2AxisX.commands.stop := #_w1;
   "Unit1.Em4.HmiInterface".cmAnodeMainPnP1AxisY.commands.stop := #_w1;
   "Unit1.Em4.HmiInterface".cmAnodeMainPnP1AxisZ.commands.stop := #_w1;
   "Unit1.Em4.HmiInterface".cmAnodeMainPnP2AxisZ.commands.stop := #_w1;
   "Unit1.Em4.HmiInterface".cmAnodeAlignTableAxisX.commands.stop := #_w1;
   "Unit1.Em4.HmiInterface".cmAnodeAlignTableAxisY1.commands.stop := #_w1;
   "Unit1.Em4.HmiInterface".cmAnodeAlignTableAxisY2.commands.stop := #_w1;
   "Unit1.Em5.HmiInterface".cmCathodeMainPnP1AxisX.commands.stop := #_w1;
   "Unit1.Em5.HmiInterface".cmCathodeMainPnP2AxisX.commands.stop := #_w1;
   "Unit1.Em5.HmiInterface".cmCathodeMainPnP1AxisY.commands.stop := #_w1;
   "Unit1.Em5.HmiInterface".cmCathodeMainPnP1AxisZ.commands.stop := #_w1;
   "Unit1.Em5.HmiInterface".cmCathodeMainPnP2AxisZ.commands.stop := #_w1;
   "Unit1.Em5.HmiInterface".cmCathodeAlignTableAxisX.commands.stop := #_w1;
   "Unit1.Em5.HmiInterface".cmCathodeAlignTableAxisY1.commands.stop := #_w1;
   "Unit1.Em5.HmiInterface".cmCathodeAlignTableAxisY2.commands.stop := #_w1;
   "Unit1.Em6.HmiInterface".cmFinalRollerFrontAxisX.commands.stop := #_w1;
   "Unit1.Em6.HmiInterface".cmFinalRollerRearAxisX.commands.stop := #_w1;
   "Unit1.Em6.HmiInterface".cmMendrelAnodeFrontAxisY.commands.stop := #_w1;
   "Unit1.Em6.HmiInterface".cmMendrelAnodeFrontAxisZ.commands.stop := #_w1;
   "Unit1.Em6.HmiInterface".cmMendrelAnodeRearAxisY.commands.stop := #_w1;
   "Unit1.Em6.HmiInterface".cmMendrelAnodeRearAxisZ.commands.stop := #_w1;
   "Unit1.Em6.HmiInterface".cmMendrelCathodeFrontAxisY.commands.stop := #_w1;
   "Unit1.Em6.HmiInterface".cmMendrelCathodeFrontAxisZ.commands.stop := #_w1;
   "Unit1.Em6.HmiInterface".cmMendrelCathodeRearAxisY.commands.stop := #_w1;
   "Unit1.Em6.HmiInterface".cmMendrelCathodeRearAxisZ.commands.stop := #_w1;
   "Unit1.Em6.HmiInterface".cmStackTableAxisZ.commands.stop := #_w1;
   "Unit1.Em6.HmiInterface".cmStackTableOutFrontAxisZ.commands.stop := #_w1;
   "Unit1.Em6.HmiInterface".cmStackTableOutRearAxisZ.commands.stop := #_w1;
   "Unit1.Em7.HmiInterface".cmSepaClampnCutterAxisX.commands.stop := #_w1;
   "Unit1.Em7.HmiInterface".cmSepaClampnCutterAxisZ.commands.stop := #_w1;
   "Unit1.Em7.HmiInterface".cmSepaGripperAxisX.commands.stop := #_w1;
   "Unit1.Em7.HmiInterface".cmSepaGripperAxisZ.commands.stop := #_w1;
   "Unit1.Em7.HmiInterface".cmSepaGripperAxisC.commands.stop := #_w1;
   "Unit1.Em7.HmiInterface".cmJRWinderRearAxisY.commands.stop := #_w1;
   "Unit1.Em7.HmiInterface".cmJRWinderFrontAxisY.commands.stop := #_w1;
   "Unit1.Em7.HmiInterface".cmJRWinderAxisB.commands.stop := #_w1;
   "Unit1.Em7.HmiInterface".cmJRPusherAxisZ.commands.stop := #_w1;
END_REGION

REGION Network 2 (SCL): Equipment Module 0 Cms Mapping
   REGION Input Mapping
       // Axis
       "ManualOperationControl_U1Em0".axis64Pos[6].monitoring := "Unit1.Em0.HmiInterface".cmUnwinderTopAxisB.monitoring;

       "ManualOperationControl_U1Em0".axis64Pos[6].configuration := "Unit1.Em0.HmiInterface".cmUnwinderTopAxisB.configuration;
       // SoftCam
       "ManualOperationControl_U1Em0".softCam[6] := "Unit1.Em0.HmiInterface".cm.softCam.unwinderTopAxisB;

       // TwoWayActuator
       "ManualOperationControl_U1Em0".twoWayActuator[1].monitoring := "Unit1.Em0.HmiInterface".cmAirShaftTopOnOff.monitoring;
   END_REGION


   REGION Output Mapping
       // Axis
       "CallManualOperationLines_ServoPos64Commands"(ManualOperationControl := "ManualOperationControl_U1Em0".axis64Pos[6].commands,
                                                     HmiInterface => "Unit1.Em0.HmiInterface".cmUnwinderTopAxisB.commands);

       // TwoWayActuator
       "Unit1.Em0.HmiInterface".cmAirShaftTopOnOff.commands := "ManualOperationControl_U1Em0".twoWayActuator[1].commands;
   END_REGION
END_REGION

REGION Network 3: Equipment Module 0
   RUNG wire#powerrail
      "CallManualOperationLines_EM"(disableUnit := #disableUnit1, manualOperationEm := "ManualOperationControl_U1Em0".manualOperationEm, manualOperationEmArea := "ManualOperationControl_U1Em0".manualOperationEmArea, manualOperationCms := "ManualOperationControl_U1Em0".manualOperationCms, Axis := "ManualOperationControl_U1Em0".axis, Axis64Pos := "ManualOperationControl_U1Em0".axis64Pos, AxisSfotCam := "ManualOperationControl_U1Em0".softCam, twoWayAcutor := "ManualOperationControl_U1Em0".twoWayActuator, Status := #StatusEm[0].Status, errorID := #errorIDEm[0].errorID)
   END_RUNG
   // the same network as SCL:
   "CallManualOperationLines_EM"(disableUnit := #disableUnit1,
                           manualOperationEm := "ManualOperationControl_U1Em0".manualOperationEm,
                           manualOperationEmArea := "ManualOperationControl_U1Em0".manualOperationEmArea,
                           manualOperationCms := "ManualOperationControl_U1Em0".manualOperationCms,
                           Axis := "ManualOperationControl_U1Em0".axis,
                           Axis64Pos := "ManualOperationControl_U1Em0".axis64Pos,
                           AxisSfotCam := "ManualOperationControl_U1Em0".softCam,
                           twoWayAcutor := "ManualOperationControl_U1Em0".twoWayActuator,
                           Status := #StatusEm[0].Status,
                           errorID := #errorIDEm[0].errorID);
END_REGION

REGION Network 4 (SCL): Equipment Module 1 Cms Mapping
   REGION Input Mapping
       // Axis
       "ManualOperationControl_U1Em1".axis64Pos[6].monitoring := "Unit1.Em1.HmiInterface".cmUnwinderBtmAxisB.monitoring;

       "ManualOperationControl_U1Em1".axis64Pos[6].configuration := "Unit1.Em1.HmiInterface".cmUnwinderBtmAxisB.configuration;
       // SoftCam
       "ManualOperationControl_U1Em1".softCam[6] := "Unit1.Em1.HmiInterface".cm.softCam.unwinderBtmAxisB;

       // TwoWayActuator
       "ManualOperationControl_U1Em1".twoWayActuator[1].monitoring := "Unit1.Em1.HmiInterface".cmAirShaftBtmOnOff.monitoring;
   END_REGION


   REGION Output Mapping
       // Axis
       "CallManualOperationLines_ServoPos64Commands"(ManualOperationControl := "ManualOperationControl_U1Em1".axis64Pos[6].commands,
                                                     HmiInterface => "Unit1.Em1.HmiInterface".cmUnwinderBtmAxisB.commands);

       // TwoWayActuator
       "Unit1.Em0.HmiInterface".cmAirShaftTopOnOff.commands := "ManualOperationControl_U1Em0".twoWayActuator[1].commands;
   END_REGION
END_REGION

REGION Network 5: Equipment Module 1
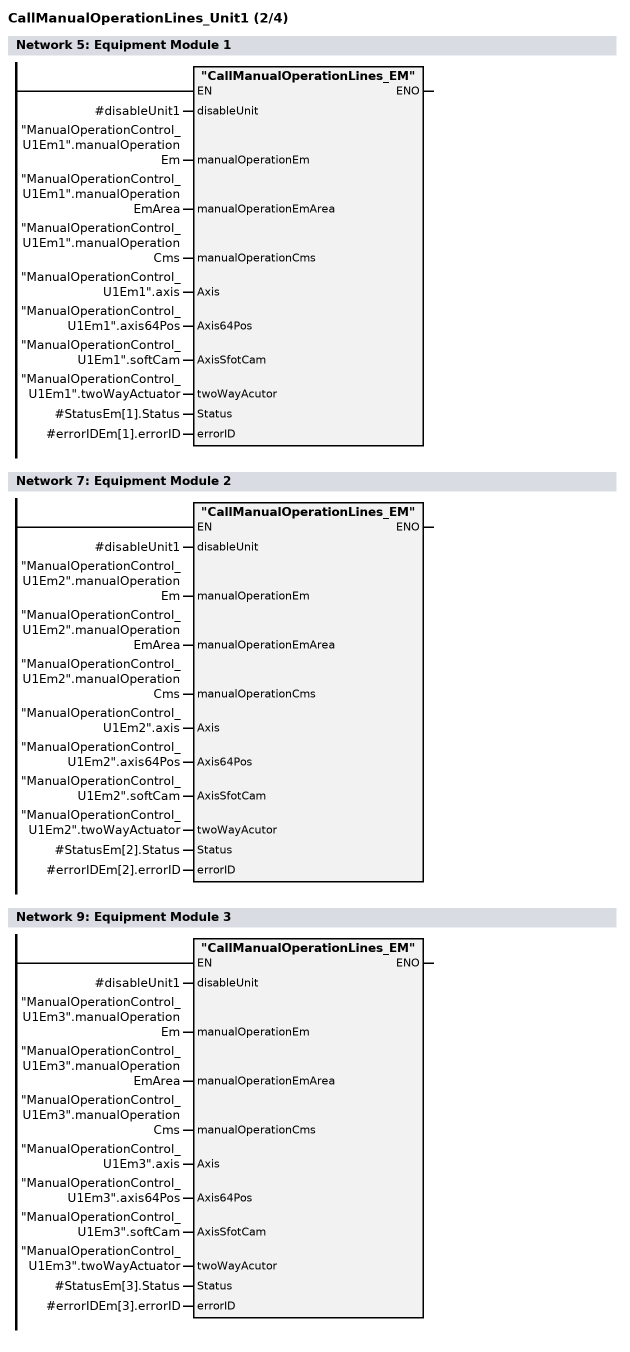
   RUNG wire#powerrail
      "CallManualOperationLines_EM"(disableUnit := #disableUnit1, manualOperationEm := "ManualOperationControl_U1Em1".manualOperationEm, manualOperationEmArea := "ManualOperationControl_U1Em1".manualOperationEmArea, manualOperationCms := "ManualOperationControl_U1Em1".manualOperationCms, Axis := "ManualOperationControl_U1Em1".axis, Axis64Pos := "ManualOperationControl_U1Em1".axis64Pos, AxisSfotCam := "ManualOperationControl_U1Em1".softCam, twoWayAcutor := "ManualOperationControl_U1Em1".twoWayActuator, Status := #StatusEm[1].Status, errorID := #errorIDEm[1].errorID)
   END_RUNG
   // the same network as SCL:
   "CallManualOperationLines_EM"(disableUnit := #disableUnit1,
                           manualOperationEm := "ManualOperationControl_U1Em1".manualOperationEm,
                           manualOperationEmArea := "ManualOperationControl_U1Em1".manualOperationEmArea,
                           manualOperationCms := "ManualOperationControl_U1Em1".manualOperationCms,
                           Axis := "ManualOperationControl_U1Em1".axis,
                           Axis64Pos := "ManualOperationControl_U1Em1".axis64Pos,
                           AxisSfotCam := "ManualOperationControl_U1Em1".softCam,
                           twoWayAcutor := "ManualOperationControl_U1Em1".twoWayActuator,
                           Status := #StatusEm[1].Status,
                           errorID := #errorIDEm[1].errorID);
END_REGION

REGION Network 6 (SCL): Equipment Module 2 Cms Mapping
   REGION Input Mapping  
       // TwoWayActuator
       "ManualOperationControl_U1Em2".twoWayActuator[1].monitoring := "Unit1.Em2.HmiInterface".cmSuctionPadTopUpDown.monitoring;
       "ManualOperationControl_U1Em2".twoWayActuator[2].monitoring := "Unit1.Em2.HmiInterface".cmSuctionPadBtmUpDown.monitoring;
       "ManualOperationControl_U1Em2".twoWayActuator[3].monitoring := "Unit1.Em2.HmiInterface".cmCutterUpDown.monitoring;
       "ManualOperationControl_U1Em2".twoWayActuator[4].monitoring := "Unit1.Em2.HmiInterface".cmTapeTopUpDown.monitoring;
       "ManualOperationControl_U1Em2".twoWayActuator[5].monitoring := "Unit1.Em2.HmiInterface".cmTapeBtmUpDown.monitoring;
       "ManualOperationControl_U1Em2".twoWayActuator[6].monitoring := "Unit1.Em2.HmiInterface".cmSpliceHeadRotateTopFwdBwd.monitoring;
       "ManualOperationControl_U1Em2".twoWayActuator[7].monitoring := "Unit1.Em2.HmiInterface".cmSpliceHeadRotateBtmFwdBwd.monitoring;
       "ManualOperationControl_U1Em2".twoWayActuator[8].monitoring := "Unit1.Em2.HmiInterface".cmSuctionPadTopLeftVaccum.monitoring;
       "ManualOperationControl_U1Em2".twoWayActuator[9].monitoring := "Unit1.Em2.HmiInterface".cmSuctionPadTopRightVaccum.monitoring;
       "ManualOperationControl_U1Em2".twoWayActuator[10].monitoring := "Unit1.Em2.HmiInterface".cmSuctionPadBtmLeftVaccum.monitoring;
       "ManualOperationControl_U1Em2".twoWayActuator[11].monitoring := "Unit1.Em2.HmiInterface".cmSuctionPadBtmRightVaccum.monitoring;
       "ManualOperationControl_U1Em2".twoWayActuator[12].monitoring := "Unit1.Em2.HmiInterface".cmSuctionPadTopTapeVaccum.monitoring;
       "ManualOperationControl_U1Em2".twoWayActuator[13].monitoring := "Unit1.Em2.HmiInterface".cmSuctionPadBtmTapeVaccum.monitoring;

   END_REGION

   REGION Output Mapping
       // TwoWayActuator
       "Unit1.Em2.HmiInterface".cmSuctionPadTopUpDown.commands := "ManualOperationControl_U1Em2".twoWayActuator[1].commands;
       "Unit1.Em2.HmiInterface".cmSuctionPadBtmUpDown.commands := "ManualOperationControl_U1Em2".twoWayActuator[2].commands;
       "Unit1.Em2.HmiInterface".cmCutterUpDown.commands := "ManualOperationControl_U1Em2".twoWayActuator[3].commands;
       "Unit1.Em2.HmiInterface".cmTapeTopUpDown.commands := "ManualOperationControl_U1Em2".twoWayActuator[4].commands;
       "Unit1.Em2.HmiInterface".cmTapeBtmUpDown.commands := "ManualOperationControl_U1Em2".twoWayActuator[5].commands;
       "Unit1.Em2.HmiInterface".cmSpliceHeadRotateTopFwdBwd.commands := "ManualOperationControl_U1Em2".twoWayActuator[6].commands;
       "Unit1.Em2.HmiInterface".cmSpliceHeadRotateBtmFwdBwd.commands := "ManualOperationControl_U1Em2".twoWayActuator[7].commands;
       "Unit1.Em2.HmiInterface".cmSuctionPadTopLeftVaccum.commands := "ManualOperationControl_U1Em2".twoWayActuator[8].commands;
       "Unit1.Em2.HmiInterface".cmSuctionPadTopRightVaccum.commands := "ManualOperationControl_U1Em2".twoWayActuator[9].commands;
       "Unit1.Em2.HmiInterface".cmSuctionPadBtmLeftVaccum.commands := "ManualOperationControl_U1Em2".twoWayActuator[10].commands;
       "Unit1.Em2.HmiInterface".cmSuctionPadBtmRightVaccum.commands := "ManualOperationControl_U1Em2".twoWayActuator[11].commands;
       "Unit1.Em2.HmiInterface".cmSuctionPadTopTapeVaccum.commands := "ManualOperationControl_U1Em2".twoWayActuator[12].commands;
       "Unit1.Em2.HmiInterface".cmSuctionPadBtmTapeVaccum.commands := "ManualOperationControl_U1Em2".twoWayActuator[13].commands;

   END_REGION
END_REGION

REGION Network 7: Equipment Module 2
   RUNG wire#powerrail
      "CallManualOperationLines_EM"(disableUnit := #disableUnit1, manualOperationEm := "ManualOperationControl_U1Em2".manualOperationEm, manualOperationEmArea := "ManualOperationControl_U1Em2".manualOperationEmArea, manualOperationCms := "ManualOperationControl_U1Em2".manualOperationCms, Axis := "ManualOperationControl_U1Em2".axis, Axis64Pos := "ManualOperationControl_U1Em2".axis64Pos, AxisSfotCam := "ManualOperationControl_U1Em2".softCam, twoWayAcutor := "ManualOperationControl_U1Em2".twoWayActuator, Status := #StatusEm[2].Status, errorID := #errorIDEm[2].errorID)
   END_RUNG
   // the same network as SCL:
   "CallManualOperationLines_EM"(disableUnit := #disableUnit1,
                           manualOperationEm := "ManualOperationControl_U1Em2".manualOperationEm,
                           manualOperationEmArea := "ManualOperationControl_U1Em2".manualOperationEmArea,
                           manualOperationCms := "ManualOperationControl_U1Em2".manualOperationCms,
                           Axis := "ManualOperationControl_U1Em2".axis,
                           Axis64Pos := "ManualOperationControl_U1Em2".axis64Pos,
                           AxisSfotCam := "ManualOperationControl_U1Em2".softCam,
                           twoWayAcutor := "ManualOperationControl_U1Em2".twoWayActuator,
                           Status := #StatusEm[2].Status,
                           errorID := #errorIDEm[2].errorID);
END_REGION

REGION Network 8 (SCL): Equipment Module 3 Cms Mapping
   REGION Input Mapping
       // Axis
       "ManualOperationControl_U1Em3".axis64Pos[6].monitoring := "Unit1.Em3.HmiInterface".cmCompensatorAxisX.monitoring;
       //"ManualOperationControl_U1Em3".axis[2].monitoring := Unit1.Em3.HmiInterface.cmSepaFeedingRollerAxisB.monitoring;
       "ManualOperationControl_U1Em3".axis64Pos[6].configuration := "Unit1.Em3.HmiInterface".cmCompensatorAxisX.configuration;
       // SoftCam
       "ManualOperationControl_U1Em3".softCam[6] := "Unit1.Em3.HmiInterface".cm.softCam.compensatorAxisX;

       // TwoWayActuator
       "ManualOperationControl_U1Em3".twoWayActuator[1].monitoring := "Unit1.Em3.HmiInterface".cmDancerFwdBwd.monitoring;
       "ManualOperationControl_U1Em3".twoWayActuator[2].monitoring := "Unit1.Em3.HmiInterface".cmSepaUnwinderIonizerTop.monitoring;
       "ManualOperationControl_U1Em3".twoWayActuator[3].monitoring := "Unit1.Em3.HmiInterface".cmSepaUnwinderIonizerBottom.monitoring;

   END_REGION

   REGION Output Mapping
       // Axis
       "CallManualOperationLines_ServoPos64Commands"(ManualOperationControl := "ManualOperationControl_U1Em3".axis64Pos[6].commands,
                                                     HmiInterface => "Unit1.Em3.HmiInterface".cmCompensatorAxisX.commands);

       // TwoWayActuator
       "Unit1.Em3.HmiInterface".cmDancerFwdBwd.commands := "ManualOperationControl_U1Em3".twoWayActuator[1].commands;
       "Unit1.Em3.HmiInterface".cmSepaUnwinderIonizerTop.commands := "ManualOperationControl_U1Em3".twoWayActuator[2].commands;
       "Unit1.Em3.HmiInterface".cmSepaUnwinderIonizerBottom.commands := "ManualOperationControl_U1Em3".twoWayActuator[3].commands;

   END_REGION
END_REGION

REGION Network 9: Equipment Module 3
   RUNG wire#powerrail
      "CallManualOperationLines_EM"(disableUnit := #disableUnit1, manualOperationEm := "ManualOperationControl_U1Em3".manualOperationEm, manualOperationEmArea := "ManualOperationControl_U1Em3".manualOperationEmArea, manualOperationCms := "ManualOperationControl_U1Em3".manualOperationCms, Axis := "ManualOperationControl_U1Em3".axis, Axis64Pos := "ManualOperationControl_U1Em3".axis64Pos, AxisSfotCam := "ManualOperationControl_U1Em3".softCam, twoWayAcutor := "ManualOperationControl_U1Em3".twoWayActuator, Status := #StatusEm[3].Status, errorID := #errorIDEm[3].errorID)
   END_RUNG
   // the same network as SCL:
   "CallManualOperationLines_EM"(disableUnit := #disableUnit1,
                           manualOperationEm := "ManualOperationControl_U1Em3".manualOperationEm,
                           manualOperationEmArea := "ManualOperationControl_U1Em3".manualOperationEmArea,
                           manualOperationCms := "ManualOperationControl_U1Em3".manualOperationCms,
                           Axis := "ManualOperationControl_U1Em3".axis,
                           Axis64Pos := "ManualOperationControl_U1Em3".axis64Pos,
                           AxisSfotCam := "ManualOperationControl_U1Em3".softCam,
                           twoWayAcutor := "ManualOperationControl_U1Em3".twoWayActuator,
                           Status := #StatusEm[3].Status,
                           errorID := #errorIDEm[3].errorID);
END_REGION

REGION Network 10 (SCL): Equipment Module 4 Cms Mapping
   REGION Input Mapping
       // Axis
       "ManualOperationControl_U1Em4".axis64Pos[6].monitoring := "Unit1.Em4.HmiInterface".cmAnodeMainPnP1AxisX.monitoring;
       "ManualOperationControl_U1Em4".axis64Pos[7].monitoring := "Unit1.Em4.HmiInterface".cmAnodeMainPnP2AxisX.monitoring;
       "ManualOperationControl_U1Em4".axis64Pos[8].monitoring := "Unit1.Em4.HmiInterface".cmAnodeMainPnP1AxisY.monitoring;
       "ManualOperationControl_U1Em4".axis64Pos[9].monitoring := "Unit1.Em4.HmiInterface".cmAnodeMainPnP1AxisZ.monitoring;
       "ManualOperationControl_U1Em4".axis64Pos[10].monitoring := "Unit1.Em4.HmiInterface".cmAnodeMainPnP2AxisZ.monitoring;
       "ManualOperationControl_U1Em4".axis64Pos[11].monitoring := "Unit1.Em4.HmiInterface".cmAnodeAlignTableAxisX.monitoring;
       "ManualOperationControl_U1Em4".axis64Pos[12].monitoring := "Unit1.Em4.HmiInterface".cmAnodeAlignTableAxisY1.monitoring;
       "ManualOperationControl_U1Em4".axis64Pos[13].monitoring := "Unit1.Em4.HmiInterface".cmAnodeAlignTableAxisY2.monitoring;

       "ManualOperationControl_U1Em4".axis64Pos[6].configuration := "Unit1.Em4.HmiInterface".cmAnodeMainPnP1AxisX.configuration;
       "ManualOperationControl_U1Em4".axis64Pos[7].configuration := "Unit1.Em4.HmiInterface".cmAnodeMainPnP2AxisX.configuration;
       "ManualOperationControl_U1Em4".axis64Pos[8].configuration := "Unit1.Em4.HmiInterface".cmAnodeMainPnP1AxisY.configuration;
       "ManualOperationControl_U1Em4".axis64Pos[9].configuration := "Unit1.Em4.HmiInterface".cmAnodeMainPnP1AxisZ.configuration;
       "ManualOperationControl_U1Em4".axis64Pos[10].configuration := "Unit1.Em4.HmiInterface".cmAnodeMainPnP2AxisZ.configuration;
       "ManualOperationControl_U1Em4".axis64Pos[11].configuration := "Unit1.Em4.HmiInterface".cmAnodeAlignTableAxisX.configuration;
       "ManualOperationControl_U1Em4".axis64Pos[12].configuration := "Unit1.Em4.HmiInterface".cmAnodeAlignTableAxisY1.configuration;
       "ManualOperationControl_U1Em4".axis64Pos[13].configuration := "Unit1.Em4.HmiInterface".cmAnodeAlignTableAxisY2.configuration;

       // SoftCam
       "ManualOperationControl_U1Em4".softCam[6] := "Unit1.Em4.HmiInterface".cm.softCam.anodeMainPnP1AxisX;
       "ManualOperationControl_U1Em4".softCam[7] := "Unit1.Em4.HmiInterface".cm.softCam.anodeMainPnP2AxisX;
       "ManualOperationControl_U1Em4".softCam[8] := "Unit1.Em4.HmiInterface".cm.softCam.anodeMainPnP1AxisY;
       "ManualOperationControl_U1Em4".softCam[9] := "Unit1.Em4.HmiInterface".cm.softCam.anodeMainPnP1AxisZ;
       "ManualOperationControl_U1Em4".softCam[10] := "Unit1.Em4.HmiInterface".cm.softCam.anodeMainPnP2AxisZ;
       "ManualOperationControl_U1Em4".softCam[11] := "Unit1.Em4.HmiInterface".cm.softCam.anodeAlignTableAxisX;
       "ManualOperationControl_U1Em4".softCam[12] := "Unit1.Em4.HmiInterface".cm.softCam.anodeAlignTableAxisY1;
       "ManualOperationControl_U1Em4".softCam[13] := "Unit1.Em4.HmiInterface".cm.softCam.anodeAlignTableAxisY2;

       // TwoWayActuator
       "ManualOperationControl_U1Em4".twoWayActuator[1].monitoring := "Unit1.Em4.HmiInterface".cmAnodeMainPnP1RotaryCwCcw.monitoring;
       "ManualOperationControl_U1Em4".twoWayActuator[2].monitoring := "Unit1.Em4.HmiInterface".cmAnodeMainPnP1SuctionPlateVacuum.monitoring;
       "ManualOperationControl_U1Em4".twoWayActuator[3].monitoring := "Unit1.Em4.HmiInterface".cmAnodeMainPnP2SuctionPlateVacuum.monitoring;
       "ManualOperationControl_U1Em4".twoWayActuator[4].monitoring := "Unit1.Em4.HmiInterface".cmAnodeAlignTableSuctionPlateVacuum.monitoring;
       "ManualOperationControl_U1Em4".twoWayActuator[5].monitoring := "Unit1.Em4.HmiInterface".cmAnodeGlassCleaning.monitoring;
       "ManualOperationControl_U1Em4".twoWayActuator[6].monitoring := "Unit1.Em4.HmiInterface".cmAnodeNgPnpUpDown.monitoring;
       "ManualOperationControl_U1Em4".twoWayActuator[7].monitoring := "Unit1.Em4.HmiInterface".cmAnodeNgPnp1stFwdBwd.monitoring;
       "ManualOperationControl_U1Em4".twoWayActuator[8].monitoring := "Unit1.Em4.HmiInterface".cmAnodeNgPnp2ndFwdBwd.monitoring;
       "ManualOperationControl_U1Em4".twoWayActuator[9].monitoring := "Unit1.Em4.HmiInterface".cmAnodeMaintenanceMovingFixFrontRearFwdBwd.monitoring;
       "ManualOperationControl_U1Em4".twoWayActuator[10].monitoring := "Unit1.Em4.HmiInterface".cmAnodeNgBoxLiftUpDown.monitoring;
       "ManualOperationControl_U1Em4".twoWayActuator[11].monitoring := "Unit1.Em4.HmiInterface".cmAnodeNgBoxLockUpDown.monitoring;
       "ManualOperationControl_U1Em4".twoWayActuator[12].monitoring := "Unit1.Em4.HmiInterface".cmAnodeNgPnpVaccum.monitoring;
       "ManualOperationControl_U1Em4".twoWayActuator[13].monitoring := "Unit1.Em4.HmiInterface".cmAnodeConveyorCoverFwdBwd.monitoring;

   END_REGION


   REGION Output Mapping
       // Axis

       "CallManualOperationLines_ServoPos64Commands"(ManualOperationControl := "ManualOperationControl_U1Em4".axis64Pos[6].commands,
                                                     HmiInterface => "Unit1.Em4.HmiInterface".cmAnodeMainPnP1AxisX.commands);

       "CallManualOperationLines_ServoPos64Commands"(ManualOperationControl := "ManualOperationControl_U1Em4".axis64Pos[7].commands,
                                                     HmiInterface => "Unit1.Em4.HmiInterface".cmAnodeMainPnP2AxisX.commands);

       "CallManualOperationLines_ServoPos64Commands"(ManualOperationControl := "ManualOperationControl_U1Em4".axis64Pos[8].commands,
                                                     HmiInterface => "Unit1.Em4.HmiInterface".cmAnodeMainPnP1AxisY.commands);

       "CallManualOperationLines_ServoPos64Commands"(ManualOperationControl := "ManualOperationControl_U1Em4".axis64Pos[9].commands,
                                                     HmiInterface => "Unit1.Em4.HmiInterface".cmAnodeMainPnP1AxisZ.commands);

       "CallManualOperationLines_ServoPos64Commands"(ManualOperationControl := "ManualOperationControl_U1Em4".axis64Pos[10].commands,
                                                     HmiInterface => "Unit1.Em4.HmiInterface".cmAnodeMainPnP2AxisZ.commands);

       "CallManualOperationLines_ServoPos64Commands"(ManualOperationControl := "ManualOperationControl_U1Em4".axis64Pos[11].commands,
                                                     HmiInterface => "Unit1.Em4.HmiInterface".cmAnodeAlignTableAxisX.commands);

       "CallManualOperationLines_ServoPos64Commands"(ManualOperationControl := "ManualOperationControl_U1Em4".axis64Pos[12].commands,
                                                     HmiInterface => "Unit1.Em4.HmiInterface".cmAnodeAlignTableAxisY1.commands);

       "CallManualOperationLines_ServoPos64Commands"(ManualOperationControl := "ManualOperationControl_U1Em4".axis64Pos[13].commands,
                                                     HmiInterface => "Unit1.Em4.HmiInterface".cmAnodeAlignTableAxisY2.commands);

       // TwoWayActuator
       "Unit1.Em4.HmiInterface".cmAnodeMainPnP1RotaryCwCcw.commands := "ManualOperationControl_U1Em4".twoWayActuator[1].commands;
       "Unit1.Em4.HmiInterface".cmAnodeMainPnP1SuctionPlateVacuum.commands := "ManualOperationControl_U1Em4".twoWayActuator[2].commands;
       "Unit1.Em4.HmiInterface".cmAnodeMainPnP2SuctionPlateVacuum.commands := "ManualOperationControl_U1Em4".twoWayActuator[3].commands;
       "Unit1.Em4.HmiInterface".cmAnodeAlignTableSuctionPlateVacuum.commands := "ManualOperationControl_U1Em4".twoWayActuator[4].commands;
       "Unit1.Em4.HmiInterface".cmAnodeGlassCleaning.commands := "ManualOperationControl_U1Em4".twoWayActuator[5].commands;
       "Unit1.Em4.HmiInterface".cmAnodeNgPnpUpDown.commands := "ManualOperationControl_U1Em4".twoWayActuator[6].commands;
       "Unit1.Em4.HmiInterface".cmAnodeNgPnp1stFwdBwd.commands := "ManualOperationControl_U1Em4".twoWayActuator[7].commands;
       "Unit1.Em4.HmiInterface".cmAnodeNgPnp2ndFwdBwd.commands := "ManualOperationControl_U1Em4".twoWayActuator[8].commands;
       "Unit1.Em4.HmiInterface".cmAnodeMaintenanceMovingFixFrontRearFwdBwd.commands := "ManualOperationControl_U1Em4".twoWayActuator[9].commands;
       "Unit1.Em4.HmiInterface".cmAnodeNgBoxLiftUpDown.commands := "ManualOperationControl_U1Em4".twoWayActuator[10].commands;
       "Unit1.Em4.HmiInterface".cmAnodeNgBoxLockUpDown.commands := "ManualOperationControl_U1Em4".twoWayActuator[11].commands;
       "Unit1.Em4.HmiInterface".cmAnodeNgPnpVaccum.commands := "ManualOperationControl_U1Em4".twoWayActuator[12].commands;
       "Unit1.Em4.HmiInterface".cmAnodeConveyorCoverFwdBwd.commands := "ManualOperationControl_U1Em4".twoWayActuator[13].commands;

   END_REGION
END_REGION

REGION Network 11: Equipment Module 4
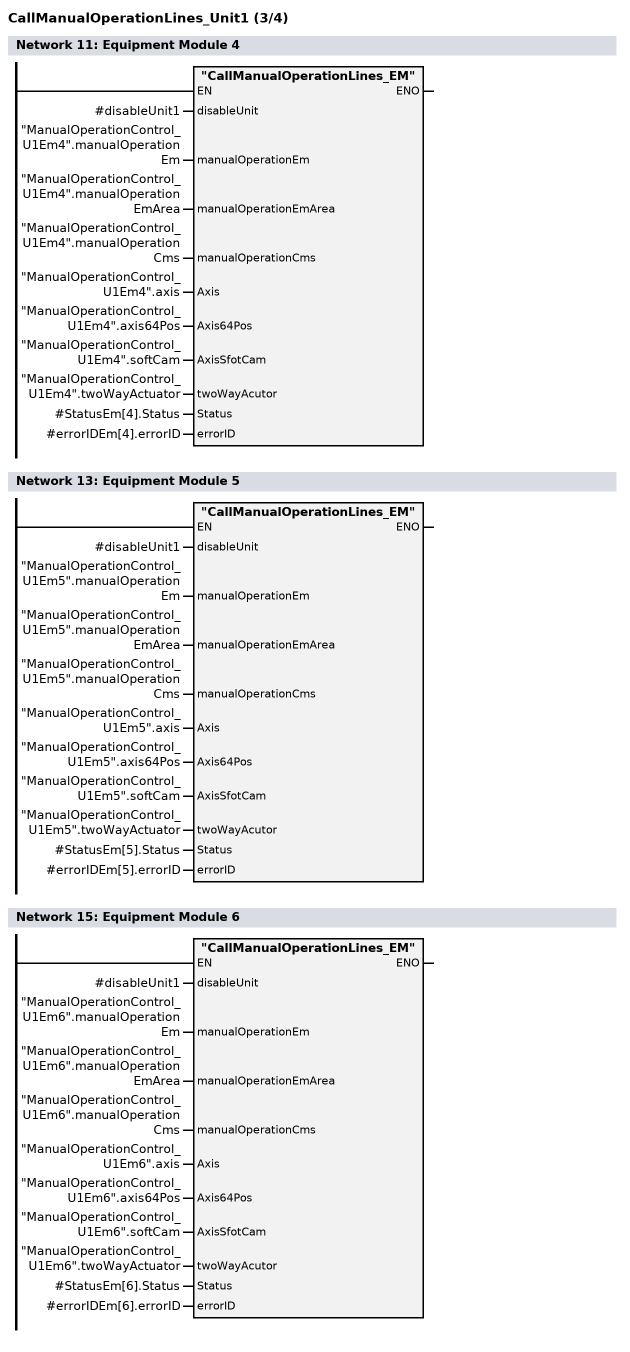
   RUNG wire#powerrail
      "CallManualOperationLines_EM"(disableUnit := #disableUnit1, manualOperationEm := "ManualOperationControl_U1Em4".manualOperationEm, manualOperationEmArea := "ManualOperationControl_U1Em4".manualOperationEmArea, manualOperationCms := "ManualOperationControl_U1Em4".manualOperationCms, Axis := "ManualOperationControl_U1Em4".axis, Axis64Pos := "ManualOperationControl_U1Em4".axis64Pos, AxisSfotCam := "ManualOperationControl_U1Em4".softCam, twoWayAcutor := "ManualOperationControl_U1Em4".twoWayActuator, Status := #StatusEm[4].Status, errorID := #errorIDEm[4].errorID)
   END_RUNG
   // the same network as SCL:
   "CallManualOperationLines_EM"(disableUnit := #disableUnit1,
                           manualOperationEm := "ManualOperationControl_U1Em4".manualOperationEm,
                           manualOperationEmArea := "ManualOperationControl_U1Em4".manualOperationEmArea,
                           manualOperationCms := "ManualOperationControl_U1Em4".manualOperationCms,
                           Axis := "ManualOperationControl_U1Em4".axis,
                           Axis64Pos := "ManualOperationControl_U1Em4".axis64Pos,
                           AxisSfotCam := "ManualOperationControl_U1Em4".softCam,
                           twoWayAcutor := "ManualOperationControl_U1Em4".twoWayActuator,
                           Status := #StatusEm[4].Status,
                           errorID := #errorIDEm[4].errorID);
END_REGION

REGION Network 12 (SCL): Equipment Module 5 Cms Mapping
   REGION Input Mapping
       // Axis
       "ManualOperationControl_U1Em5".axis64Pos[6].monitoring := "Unit1.Em5.HmiInterface".cmCathodeMainPnP1AxisX.monitoring;
       "ManualOperationControl_U1Em5".axis64Pos[7].monitoring := "Unit1.Em5.HmiInterface".cmCathodeMainPnP2AxisX.monitoring;
       "ManualOperationControl_U1Em5".axis64Pos[8].monitoring := "Unit1.Em5.HmiInterface".cmCathodeMainPnP1AxisY.monitoring;
       "ManualOperationControl_U1Em5".axis64Pos[9].monitoring := "Unit1.Em5.HmiInterface".cmCathodeMainPnP1AxisZ.monitoring;
       "ManualOperationControl_U1Em5".axis64Pos[10].monitoring := "Unit1.Em5.HmiInterface".cmCathodeMainPnP2AxisZ.monitoring;
       "ManualOperationControl_U1Em5".axis64Pos[11].monitoring := "Unit1.Em5.HmiInterface".cmCathodeAlignTableAxisX.monitoring;
       "ManualOperationControl_U1Em5".axis64Pos[12].monitoring := "Unit1.Em5.HmiInterface".cmCathodeAlignTableAxisY1.monitoring;
       "ManualOperationControl_U1Em5".axis64Pos[13].monitoring := "Unit1.Em5.HmiInterface".cmCathodeAlignTableAxisY2.monitoring;

       "ManualOperationControl_U1Em5".axis64Pos[6].configuration := "Unit1.Em5.HmiInterface".cmCathodeMainPnP1AxisX.configuration;
       "ManualOperationControl_U1Em5".axis64Pos[7].configuration := "Unit1.Em5.HmiInterface".cmCathodeMainPnP2AxisX.configuration;
       "ManualOperationControl_U1Em5".axis64Pos[8].configuration := "Unit1.Em5.HmiInterface".cmCathodeMainPnP1AxisY.configuration;
       "ManualOperationControl_U1Em5".axis64Pos[9].configuration := "Unit1.Em5.HmiInterface".cmCathodeMainPnP1AxisZ.configuration;
       "ManualOperationControl_U1Em5".axis64Pos[10].configuration := "Unit1.Em5.HmiInterface".cmCathodeMainPnP2AxisZ.configuration;
       "ManualOperationControl_U1Em5".axis64Pos[11].configuration := "Unit1.Em5.HmiInterface".cmCathodeAlignTableAxisX.configuration;
       "ManualOperationControl_U1Em5".axis64Pos[12].configuration := "Unit1.Em5.HmiInterface".cmCathodeAlignTableAxisY1.configuration;
       "ManualOperationControl_U1Em5".axis64Pos[13].configuration := "Unit1.Em5.HmiInterface".cmCathodeAlignTableAxisY2.configuration;
       // SoftCam
       "ManualOperationControl_U1Em5".softCam[6] := "Unit1.Em5.HmiInterface".cm.softCam.cathodeMainPnP1AxisX;
       "ManualOperationControl_U1Em5".softCam[7] := "Unit1.Em5.HmiInterface".cm.softCam.cathodeMainPnP2AxisX;
       "ManualOperationControl_U1Em5".softCam[8] := "Unit1.Em5.HmiInterface".cm.softCam.cathodeMainPnP1AxisY;
       "ManualOperationControl_U1Em5".softCam[9] := "Unit1.Em5.HmiInterface".cm.softCam.cathodeMainPnP1AxisZ;
       "ManualOperationControl_U1Em5".softCam[10] := "Unit1.Em5.HmiInterface".cm.softCam.cathodeMainPnP2AxisZ;
       "ManualOperationControl_U1Em5".softCam[11] := "Unit1.Em5.HmiInterface".cm.softCam.cathodeAlignTableAxisX;
       "ManualOperationControl_U1Em5".softCam[12] := "Unit1.Em5.HmiInterface".cm.softCam.cathodeAlignTableAxisY1;
       "ManualOperationControl_U1Em5".softCam[13] := "Unit1.Em5.HmiInterface".cm.softCam.cathodeAlignTableAxisY2;

       // TwoWayActuator
       "ManualOperationControl_U1Em5".twoWayActuator[1].monitoring := "Unit1.Em5.HmiInterface".cmCathodeMainPnP1RotaryCwCcw.monitoring;
       "ManualOperationControl_U1Em5".twoWayActuator[2].monitoring := "Unit1.Em5.HmiInterface".cmCathodeMainPnP1SuctionPlateVacuum.monitoring;
       "ManualOperationControl_U1Em5".twoWayActuator[3].monitoring := "Unit1.Em5.HmiInterface".cmCathodeMainPnP2SuctionPlateVacuum.monitoring;
       "ManualOperationControl_U1Em5".twoWayActuator[4].monitoring := "Unit1.Em5.HmiInterface".cmCathodeAlignTableSuctionPlateVacuum.monitoring;
       "ManualOperationControl_U1Em5".twoWayActuator[5].monitoring := "Unit1.Em5.HmiInterface".cmCathodeGlassCleaning.monitoring;
       "ManualOperationControl_U1Em5".twoWayActuator[6].monitoring := "Unit1.Em5.HmiInterface".cmCathodeNgPnpUpDown.monitoring;
       "ManualOperationControl_U1Em5".twoWayActuator[7].monitoring := "Unit1.Em5.HmiInterface".cmCathodeNgPnp1stFwdBwd.monitoring;
       "ManualOperationControl_U1Em5".twoWayActuator[8].monitoring := "Unit1.Em5.HmiInterface".cmCathodeNgPnp2ndFwdBwd.monitoring;
       "ManualOperationControl_U1Em5".twoWayActuator[9].monitoring := "Unit1.Em5.HmiInterface".cmCathodeMaintenanceMovingFixFrontRearFwdBwd.monitoring;
       "ManualOperationControl_U1Em5".twoWayActuator[10].monitoring := "Unit1.Em5.HmiInterface".cmCathodeNgBoxLiftUpDown.monitoring;
       "ManualOperationControl_U1Em5".twoWayActuator[11].monitoring := "Unit1.Em5.HmiInterface".cmCathodeNgBoxLockUpDown.monitoring;
       "ManualOperationControl_U1Em5".twoWayActuator[12].monitoring := "Unit1.Em5.HmiInterface".cmCathodeNgPnpVaccum.monitoring;
       "ManualOperationControl_U1Em5".twoWayActuator[13].monitoring := "Unit1.Em5.HmiInterface".cmCathodeConveyorCoverFwdBwd.monitoring;

   END_REGION


   REGION Output Mapping
       // Axis
       "CallManualOperationLines_ServoPos64Commands"(ManualOperationControl := "ManualOperationControl_U1Em5".axis64Pos[6].commands,
                                                     HmiInterface => "Unit1.Em5.HmiInterface".cmCathodeMainPnP1AxisX.commands);

